# B&R Automation Studio project NAELD004C00R10L518F00 (part 27)

#### Act_Main.st
```iecst
(** 2019-07-03 **)
ACTION Act_Main:

	IF eStatOld <> eStat THEN
		fbDirCreate1(bEn := FALSE);
		fbDirCreate2(bEn := FALSE);
		fbFileRead1(bEn := FALSE);
		fbFileWrite1(bEn := FALSE);
		usiStep	:= 0;

		bFileNotFound			:= FALSE;
		bNewProduct				:= FALSE;
		bLastProductUnload		:= FALSE;
		bLastProductLeftInBffr	:= FALSE;

		sStatTxt	:= a_sStatText[eStat];

		eStatOld	:= eStat;

		eStatus		:= Busy;
	END_IF

	//Main
	CASE eStat OF

		BufferActIdle:
			eStatus	:= Idle;

		BufferActCreateDir:
			IF eStatus = Idle OR eStatus = Busy THEN

				eStatus	:= Busy;

				CASE usiStep OF
					0:
						fbDirCreate1(bEn := TRUE);
						IF fbDirCreate1.udiStatus = 0 THEN
							usiStep	:= 1;
						ELSIF fbDirCreate1.udiStatus < 65534 THEN
							eStatus		:= Error;

							IF fbDirCreate1.udiStatus = 1908 THEN
								udiStatus	:= 10000;	//Create User Directory Error
							ELSE
								udiStatus	:= fbDirCreate1.udiStatus;
							END_IF
						END_IF

					1:
						fbDirCreate2(bEn := TRUE);
						IF fbDirCreate2.udiStatus = 0 THEN
							eStatus	:= Done;
						ELSIF fbDirCreate2.udiStatus < 65534 THEN
							eStatus		:= Error;

							IF fbDirCreate2.udiStatus = 1908 THEN
								udiStatus	:= 10001;	//Create Retain Directory Error
							ELSE
								udiStatus	:= fbDirCreate2.udiStatus;
							END_IF
						END_IF

				END_CASE

			END_IF

		BufferActGetRetainBffr:
			IF eStatus = Idle OR eStatus = Busy THEN

				eStatus	:= Busy;

				fbFileRead1(bEn := TRUE);
				IF fbFileRead1.udiStatus = 0 THEN
					eStatus	:= Done;

					tyBffrParameter.diBffrTtlSlt	:= p_diBffrTtlSlt;
					tyBffrParameter.diSltCap		:= p_diSltCap;

					fBffrStat(ADR(p_tyBufferStat) , p_tyBuffer);
					fDispBffrDescending(ADR(p_tyDispBuffer) , tyBffrParameter , p_tyBuffer , p_dtCurrDT , DINT_TO_TIME(p_diCoolTm) , 0 , 1 , 2);

				ELSIF fbFileRead1.udiStatus < 65534 THEN
					eStatus	:= Error;

					IF fbFileRead1.udiStatus = 1900 THEN
						udiStatus	:= 10002;	//File Open Error While Reading Retain File
					ELSIF fbFileRead1.udiStatus = 1902 THEN
						udiStatus	:= 10003;	//File Read Error While Reading Retain File
					ELSIF fbFileRead1.udiStatus = 1904 THEN
						udiStatus	:= 10004;	//File Close Error While Reading Retain File
					ELSIF fbFileRead1.udiStatus = 1915 THEN
						eStatus			:= Done;
						bFileNotFound	:= TRUE;
					ELSE
						udiStatus	:= fbFileRead1.udiStatus;
					END_IF
				END_IF

			END_IF

		BufferActSetFull:
			IF eStatus = Idle OR eStatus = Busy THEN

				eStatus	:= Busy;

				CASE usiStep OF
					0:
						tyBffrParameter.bAscending		:= p_bAscending;
						tyBffrParameter.diBffrTtlSlt	:= p_diBffrTtlSlt;
						tyBffrParameter.diMaxSlt		:= p_diMaxSlt;
						tyBffrParameter.diMinSlt		:= p_diMinSlt;
						tyBffrParameter.diPitch			:= p_diPitch;
						tyBffrParameter.diSltCap		:= p_diSltCap;
						tyBffrParameter.a_bSkip			:= pa_bSkip;
						bFIFOOld						:= p_bFIFO;

						udiStatus	:= fBffrSetFull(ADR(p_tyBuffer) , tyBffrParameter , p_dtCurrDT , p_sBffrNm , p_sProdNm);

						IF udiStatus = 0 THEN
							usiStep	:= 1;

							fBffrStat(ADR(p_tyBufferStat) , p_tyBuffer);
							fDispBffrDescending(ADR(p_tyDispBuffer) , tyBffrParameter , p_tyBuffer , p_dtCurrDT , DINT_TO_TIME(p_diCoolTm) , 0 , 1 , 2);

						ELSE
							eStatus	:= Error;

						END_IF

					1:
						fbFileWrite1(bEn := TRUE);

						IF fbFileWrite1.udiStatus = 0 THEN
							eStatus	:= Done;
						ELSIF fbFileWrite1.udiStatus < 65534 THEN
							eStatus	:= Error;

							IF fbFileWrite1.udiStatus = 1900 THEN
								udiStatus	:= 10005;	//File Open Error While Setting Full Buffer
							ELSIF fbFileWrite1.udiStatus = 1901 THEN
								udiStatus	:= 10006;	//File Create Error While Setting Full Buffer
							ELSIF fbFileWrite1.udiStatus = 1903 THEN
								udiStatus	:= 10007;	//File Write Error While Setting Full Buffer
							ELSIF fbFileWrite1.udiStatus = 1904 THEN
								udiStatus	:= 10008;	//File Close Error While Setting Full Buffer
							ELSIF fbFileWrite1.udiStatus = 1914 THEN
								udiStatus	:= 10040;	//Directory Does Not Exist While Setting Full Buffer
							ELSE
								udiStatus	:= fbFileWrite1.udiStatus;
							END_IF
						END_IF

				END_CASE

			END_IF

		BufferActSetMty:
			IF eStatus = Idle OR eStatus = Busy THEN

				eStatus	:= Busy;

				CASE usiStep OF
					0:
						tyBffrParameter.bAscending		:= p_bAscending;
						tyBffrParameter.diBffrTtlSlt	:= p_diBffrTtlSlt;
						tyBffrParameter.diMaxSlt		:= p_diMaxSlt;
						tyBffrParameter.diMinSlt		:= p_diMinSlt;
						tyBffrParameter.diPitch			:= p_diPitch;
						tyBffrParameter.diSltCap		:= p_diSltCap;
						tyBffrParameter.a_bSkip			:= pa_bSkip;
						bFIFOOld						:= p_bFIFO;

						udiStatus	:= fBffrSetMty(ADR(p_tyBuffer) , tyBffrParameter , p_sBffrNm);

						IF udiStatus = 0 THEN
							usiStep	:= 1;

							fBffrStat(ADR(p_tyBufferStat) , p_tyBuffer);
							fDispBffrDescending(ADR(p_tyDispBuffer) , tyBffrParameter , p_tyBuffer , p_dtCurrDT , DINT_TO_TIME(p_diCoolTm) , 0 , 1 , 2);

						ELSE
							eStatus	:= Error;

						END_IF

					1:
						fbFileWrite1(bEn := TRUE);

						IF fbFileWrite1.udiStatus = 0 THEN
							eStatus	:= Done;
						ELSIF fbFileWrite1.udiStatus < 65534 THEN
							eStatus	:= Error;

							IF fbFileWrite1.udiStatus = 1900 THEN
								udiStatus	:= 10009;	//File Open Error While Setting Empty Buffer
							ELSIF fbFileWrite1.udiStatus = 1901 THEN
								udiStatus	:= 10010;	//File Create Error While Setting Empty Buffer
							ELSIF fbFileWrite1.udiStatus = 1903 THEN
								udiStatus	:= 10011;	//File Write Error While Setting Empty Buffer
							ELSIF fbFileWrite1.udiStatus = 1904 THEN
								udiStatus	:= 10012;	//File Close Error While Setting Empty Buffer
							ELSIF fbFileWrite1.udiStatus = 1914 THEN
								udiStatus	:= 10041;	//Directory Does Not Exist While Setting Empty Buffer
							ELSE
								udiStatus	:= fbFileWrite1.udiStatus;
							END_IF
						END_IF

				END_CASE

			END_IF

		BufferActLoad:
			IF eStatus = Idle OR eStatus = Busy THEN

				eStatus	:= Busy;

				CASE usiStep OF
					0:
						diCurrSlt	:= fLifterPosInUMToSltBtmMin(p_diLifterCurrPosInUM , p_diSltToSltInUM , p_diLifterBtmPosInUM);

						udiStatus	:= fBffrLoad(ADR(p_tyBuffer) , ADR(bNewProduct) , diCurrSlt , p_dtCurrDT , p_bGdBrdIn , p_sProdNm , p_sBarcode1 , p_sBarcode2);

						IF udiStatus = 0 THEN
							usiStep	:= 1;

							tyBffrParameter.diBffrTtlSlt	:= p_diBffrTtlSlt;
							tyBffrParameter.diSltCap		:= p_diSltCap;

							fBffrStat(ADR(p_tyBufferStat) , p_tyBuffer);
							fDispBffrDescending(ADR(p_tyDispBuffer) , tyBffrParameter , p_tyBuffer , p_dtCurrDT , DINT_TO_TIME(p_diCoolTm) , 0 , 1 , 2);

						ELSE
							eStatus	:= Error;

							IF udiStatus = 1010 THEN
								udiStatus	:= 10076;	//Loading Slot Is Not For Board
							ELSIF udiStatus = 1011 THEN
								udiStatus	:= 10077;	//Loading Slot Is Full Of Board
							ELSIF udiStatus = 1012 THEN
								udiStatus	:= 10078;	//Loading First Sub-Slot Is Not For Board
							ELSIF udiStatus	= 1013 THEN
								udiStatus	:= 10079;	//Loading Last Sub-Slot Have Board, Which Mean Slot Is Full Of Board
							ELSIF udiStatus = 1014 THEN
								udiStatus	:= 10080;	//Loading Last Sub-Slot Is Not For Board
							ELSIF udiStatus = 1015 THEN
								udiStatus	:= 10081;	//Loading Slot Is Full Of Board
							ELSIF udiStatus = 1001 THEN
								udiStatus	:= 10082;	//Loading Slot Is Skipped
							ELSIF udiStatus	= 1016 THEN
								udiStatus	:= 10083;	//Existing Board Status Is Different With Loading Board Status
							END_IF

						END_IF

					1:
						fbFileWrite1(bEn := TRUE);

						IF fbFileWrite1.udiStatus = 0 THEN
							eStatus	:= Done;
						ELSIF fbFileWrite1.udiStatus < 65534 THEN
							eStatus	:= Error;

							IF fbFileWrite1.udiStatus = 1900 THEN
								udiStatus	:= 10013;	//File Open Error While Loading Info To Buffer
							ELSIF fbFileWrite1.udiStatus = 1901 THEN
								udiStatus	:= 10014;	//File Create Error While Loading Info To Buffer
							ELSIF fbFileWrite1.udiStatus = 1903 THEN
								udiStatus	:= 10015;	//File Write Error While Loading Info To Buffer
							ELSIF fbFileWrite1.udiStatus = 1904 THEN
								udiStatus	:= 10016;	//File Close Error While Loading Info To Buffer
							ELSIF fbFileWrite1.udiStatus = 1914 THEN
								udiStatus	:= 10042;	//Directory Does Not Exist While Loading Info To Buffer
							ELSE
								udiStatus	:= fbFileWrite1.udiStatus;
							END_IF
						END_IF

				END_CASE

			END_IF

		BufferActLoadSltChk:
			IF eStatus = Idle OR eStatus = Busy THEN

				eStatus	:= Busy;

				CASE usiStep OF
					0:
						diCurrSlt	:= fLifterPosInUMToSltBtmMin(p_diLifterCurrPosInUM , p_diSltToSltInUM , p_diLifterBtmPosInUM);

						IF p_bNxtLoadSeq = TRUE AND p_bGdBrdIn = TRUE THEN
							diExpectedSlt	:= fBffrNxtLoadSeqGd(p_bAscending , p_tyBuffer);
						ELSIF p_bNxtLoadSeq = TRUE AND p_bGdBrdIn = FALSE THEN
							diExpectedSlt	:= fBffrNxtLoadSeqBad(p_bAscending , p_tyBuffer);
						ELSIF p_bNxtLoadSeq = FALSE AND p_bGdBrdIn = TRUE THEN
							diExpectedSlt	:= fBffrNxtLoadNearbyGd(diCurrSlt , p_tyBuffer);
						ELSE
							diExpectedSlt	:= fBffrNxtLoadNearbyBad(diCurrSlt , p_tyBuffer);
						END_IF

						IF diCurrSlt = diExpectedSlt THEN
							udiStatus	:= fBffrLoad(ADR(p_tyBuffer) , ADR(bNewProduct) , diCurrSlt , p_dtCurrDT , p_bGdBrdIn , p_sProdNm , p_sBarcode1 , p_sBarcode2);

							IF udiStatus = 0 THEN
								usiStep	:= 1;

								tyBffrParameter.diBffrTtlSlt	:= p_diBffrTtlSlt;
								tyBffrParameter.diSltCap		:= p_diSltCap;

								fBffrStat(ADR(p_tyBufferStat) , p_tyBuffer);
								fDispBffrDescending(ADR(p_tyDispBuffer) , tyBffrParameter , p_tyBuffer , p_dtCurrDT , DINT_TO_TIME(p_diCoolTm) , 0 , 1 , 2);

							ELSE
								eStatus	:= Error;

								IF udiStatus = 1010 THEN
									udiStatus	:= 10084;	//Loading Slot Is Not For Board
								ELSIF udiStatus = 1011 THEN
									udiStatus	:= 10085;	//Loading Slot Is Full Of Board
								ELSIF udiStatus = 1012 THEN
									udiStatus	:= 10086;	//Loading First Sub-Slot Is Not For Board
								ELSIF udiStatus	= 1013 THEN
									udiStatus	:= 10087;	//Loading Last Sub-Slot Have Board, Which Mean Slot Is Full Of Board
								ELSIF udiStatus = 1014 THEN
									udiStatus	:= 10088;	//Loading Last Sub-Slot Is Not For Board
								ELSIF udiStatus = 1015 THEN
									udiStatus	:= 10089;	//Loading Slot Is Full Of Board
								ELSIF udiStatus = 1001 THEN
									udiStatus	:= 10090;	//Loading Slot Is Skipped
								ELSIF udiStatus	= 1016 THEN
									udiStatus	:= 10091;	//Existing Board Status Is Different With Loading Board Status
								END_IF

							END_IF

						ELSE
							udiStatus	:= 10017;	//Wrong Slot Number To Load
							eStatus		:= Error;

						END_IF

					1:
						fbFileWrite1(bEn := TRUE);

						IF fbFileWrite1.udiStatus = 0 THEN
							eStatus	:= Done;
						ELSIF fbFileWrite1.udiStatus < 65534 THEN
							eStatus	:= Error;

							IF fbFileWrite1.udiStatus = 1900 THEN
								udiStatus	:= 10018;	//File Open Error While Loading Info To Buffer With Slot Check
							ELSIF fbFileWrite1.udiStatus = 1901 THEN
								udiStatus	:= 10019;	//File Create Error While Loading Info To Buffer With Slot Check
							ELSIF fbFileWrite1.udiStatus = 1903 THEN
								udiStatus	:= 10020;	//File Write Error While Loading Info To Buffer With Slot Check
							ELSIF fbFileWrite1.udiStatus = 1904 THEN
								udiStatus	:= 10021;	//File Close Error While Loading Info To Buffer With Slot Check
							ELSIF fbFileWrite1.udiStatus = 1914 THEN
								udiStatus	:= 10043;	//Directory Does Not Exist While Loading Info To Buffer With Slot Check
							ELSE
								udiStatus	:= fbFileWrite1.udiStatus;
							END_IF
						END_IF

				END_CASE

			END_IF

		BufferActUnload:
			IF eStatus = Idle OR eStatus = Busy THEN

				eStatus	:= Busy;

				CASE usiStep OF
					0:
						IF p_bLinkMcParamProdSelTopToBtm  AND p_bLinkProjLifterMagPlatform = FALSE THEN //TravLif with Top to Btm
							diCurrSlt	:= fLifterPosInUMToSltTopMin(p_diLifterCurrPosInUM , p_diSltToSltInUM , p_diLifterBtmPosInUM);
						ELSE
							diCurrSlt	:= fLifterPosInUMToSltBtmMin(p_diLifterCurrPosInUM , p_diSltToSltInUM , p_diLifterBtmPosInUM);
						END_IF

						udiStatus	:= fBffrUnload(ADR(tyBoardUnloadStat) , ADR(p_tyBuffer) , ADR(bLastProductUnload) , ADR(bLastProductLeftInBffr) , diCurrSlt);

						IF p_sCurrRcpNm = tyBoardUnloadStat.sProdNm THEN
							bLastProductUnload	:= FALSE;
						END_IF

						IF udiStatus = 0 THEN
							usiStep	:= 1;

							tyBffrParameter.diBffrTtlSlt	:= p_diBffrTtlSlt;
							tyBffrParameter.diSltCap		:= p_diSltCap;

							fBffrStat(ADR(p_tyBufferStat) , p_tyBuffer);
							fDispBffrDescending(ADR(p_tyDispBuffer) , tyBffrParameter , p_tyBuffer , p_dtCurrDT , DINT_TO_TIME(p_diCoolTm) , 0 , 1 , 2);

						ELSE
							eStatus	:= Error;

							IF udiStatus = 1000 THEN
								udiStatus	:= 10048;	//Unloading Slot Is Skipped While Unloading Buffer
							ELSIF udiStatus = 1003 THEN
								udiStatus	:= 10049;	//Unloading Slot Is Not For Board While Unloading Buffer
							ELSIF udiStatus = 1004 THEN
								udiStatus	:= 10050;	//Unloading Slot Board Is Not available While Unloading Buffer
							ELSIF udiStatus = 1005 THEN
								udiStatus	:= 10051;	//Unloading Last Sub Slot Is Not For Board While Unloading Buffer
							ELSIF udiStatus = 1006 THEN
								udiStatus	:= 10052;	//Unloading Last Sub Slot Has No Board While Unloading Buffer
							ELSIF udiStatus = 1007 THEN
								udiStatus	:= 10053;	//Board Quantity In Slot Is 0 While Unloading Buffer
							ELSIF udiStatus = 1008 THEN
								udiStatus	:= 10054;	//Board Capacity In Slot Is 0 While Unloading Buffer
							END_IF

						END_IF

					1:
						fbFileWrite1(bEn := TRUE);

						IF fbFileWrite1.udiStatus = 0 THEN
							eStatus	:= Done;
						ELSIF fbFileWrite1.udiStatus < 65534 THEN
							eStatus	:= Error;

							IF fbFileWrite1.udiStatus = 1900 THEN
								udiStatus	:= 10022;	//File Open Error While Unloading Info From Buffer
							ELSIF fbFileWrite1.udiStatus = 1901 THEN
								udiStatus	:= 10023;	//File Create Error While Unloading Info From Buffer
							ELSIF fbFileWrite1.udiStatus = 1903 THEN
								udiStatus	:= 10024;	//File Write Error While Unloading Info From Buffer
							ELSIF fbFileWrite1.udiStatus = 1904 THEN
								udiStatus	:= 10025;	//File Close Error While Unloading Info From Buffer
							ELSIF fbFileWrite1.udiStatus = 1914 THEN
								udiStatus	:= 10044;	//Directory Does Not Exist While Unloading Info From Buffer
							ELSE
								udiStatus	:= fbFileWrite1.udiStatus;
							END_IF
						END_IF

				END_CASE

			END_IF

		BufferActUnloadSltChk:
			IF eStatus = Idle OR eStatus = Busy THEN

				eStatus	:= Busy;

				CASE usiStep OF
					0:
						diCurrSlt	:= fLifterPosInUMToSltBtmMin(p_diLifterCurrPosInUM , p_diSltToSltInUM , p_diLifterBtmPosInUM);

						IF p_bFIFO = TRUE AND p_bGdBrdReq = TRUE THEN
							diExpectedSlt	:= fBffrNxtUnloadFIFOGd(p_tyBuffer , '');
						ELSIF p_bFIFO = TRUE AND p_bGdBrdReq = FALSE THEN
							diExpectedSlt	:= fBffrNxtUnloadFIFOBad(p_tyBuffer , '');
						ELSIF p_bFIFO = FALSE AND p_bGdBrdReq = TRUE THEN
							diExpectedSlt	:= fBffrNxtUnloadLIFOGd(p_tyBuffer , '');
						ELSE
							diExpectedSlt	:= fBffrNxtUnloadLIFOBad(p_tyBuffer , '');
						END_IF

						IF diCurrSlt = diExpectedSlt THEN
							udiStatus	:= fBffrUnload(ADR(tyBoardUnloadStat) , ADR(p_tyBuffer) , ADR(bLastProductUnload) , ADR(bLastProductLeftInBffr) , diCurrSlt);

							IF p_sCurrRcpNm = tyBoardUnloadStat.sProdNm THEN
								bLastProductUnload	:= FALSE;
							END_IF

							IF udiStatus = 0 THEN
								usiStep	:= 1;

								tyBffrParameter.diBffrTtlSlt	:= p_diBffrTtlSlt;
								tyBffrParameter.diSltCap		:= p_diSltCap;

								fBffrStat(ADR(p_tyBufferStat) , p_tyBuffer);
								fDispBffrDescending(ADR(p_tyDispBuffer) , tyBffrParameter , p_tyBuffer , p_dtCurrDT , DINT_TO_TIME(p_diCoolTm) , 0 , 1 , 2);

							ELSE
								eStatus	:= Error;

								IF udiStatus = 1000 THEN
									udiStatus	:= 10055;	//Unloading Slot Is Skipped While Unloading Buffer With Slot Check
								ELSIF udiStatus = 1003 THEN
									udiStatus	:= 10056;	//Unloading Slot Is Not For Board While Unloading Buffer With Slot Check
								ELSIF udiStatus = 1004 THEN
									udiStatus	:= 10057;	//Unloading Slot Board Is Not available While Unloading Buffer With Slot Check
								ELSIF udiStatus = 1005 THEN
									udiStatus	:= 10058;	//Unloading Last Sub Slot Is Not For Board While Unloading Buffer With Slot Check
								ELSIF udiStatus = 1006 THEN
									udiStatus	:= 10059;	//Unloading Last Sub Slot Has No Board While Unloading Buffer With Slot Check
								ELSIF udiStatus = 1007 THEN
									udiStatus	:= 10060;	//Board Quantity In Slot Is 0 While Unloading Buffer With Slot Check
								ELSIF udiStatus = 1008 THEN
									udiStatus	:= 10061;	//Board Capacity In Slot Is 0 While Unloading Buffer With Slot Check
								END_IF

							END_IF

						ELSE
							udiStatus	:= 10026;	//Wrong Slot Number To Unload
							eStatus		:= Error;

						END_IF

					1:
						fbFileWrite1(bEn := TRUE);

						IF fbFileWrite1.udiStatus = 0 THEN
							eStatus	:= Done;
						ELSIF fbFileWrite1.udiStatus < 65534 THEN
							eStatus	:= Error;

							IF fbFileWrite1.udiStatus = 1900 THEN
								udiStatus	:= 10027;	//File Open Error While Unloading Info From Buffer With Slot Check
							ELSIF fbFileWrite1.udiStatus = 1901 THEN
								udiStatus	:= 10028;	//File Create Error While Unloading Info From Buffer With Slot Check
							ELSIF fbFileWrite1.udiStatus = 1903 THEN
								udiStatus	:= 10029;	//File Write Error While Unloading Info From Buffer With Slot Check
							ELSIF fbFileWrite1.udiStatus = 1904 THEN
								udiStatus	:= 10030;	//File Close Error While Unloading Info From Buffer With Slot Check
							ELSIF fbFileWrite1.udiStatus = 1914 THEN
								udiStatus	:= 10045;	//Directory Does Not Exist While Unloading Info From Buffer With Slot Check
							ELSE
								udiStatus	:= fbFileWrite1.udiStatus;
							END_IF
						END_IF

				END_CASE

			END_IF

		BufferActUnloadCoolChk:
			IF eStatus = Idle OR eStatus = Busy THEN

				eStatus	:= Busy;

				CASE usiStep OF
					0:
						diCurrSlt	:= fLifterPosInUMToSltBtmMin(p_diLifterCurrPosInUM , p_diSltToSltInUM , p_diLifterBtmPosInUM);

						bCoolNotRdy	:= NOT fBffrChkCoolTmRdy(diCurrSlt, p_dtCurrDT, DINT_TO_TIME(p_diCoolTm), p_tyBuffer);

						IF bCoolNotRdy = FALSE THEN
							udiStatus	:= fBffrUnload(ADR(tyBoardUnloadStat) , ADR(p_tyBuffer) , ADR(bLastProductUnload) , ADR(bLastProductLeftInBffr) , diCurrSlt);

							IF p_sCurrRcpNm = tyBoardUnloadStat.sProdNm THEN
								bLastProductUnload	:= FALSE;
							END_IF

							IF udiStatus = 0 THEN
								usiStep	:= 1;

								tyBffrParameter.diBffrTtlSlt	:= p_diBffrTtlSlt;
								tyBffrParameter.diSltCap		:= p_diSltCap;

								fBffrStat(ADR(p_tyBufferStat) , p_tyBuffer);
								fDispBffrDescending(ADR(p_tyDispBuffer) , tyBffrParameter , p_tyBuffer , p_dtCurrDT , DINT_TO_TIME(p_diCoolTm) , 0 , 1 , 2);

							ELSE
								eStatus	:= Error;

								IF udiStatus = 1000 THEN
									udiStatus	:= 10062;	//Unloading Slot Is Skipped While Unloading Buffer With Cool Check
								ELSIF udiStatus = 1003 THEN
									udiStatus	:= 10063;	//Unloading Slot Is Not For Board While Unloading Buffer With Cool Check
								ELSIF udiStatus = 1004 THEN
									udiStatus	:= 10064;	//Unloading Slot Board Is Not available While Unloading Buffer With Cool Check
								ELSIF udiStatus = 1005 THEN
									udiStatus	:= 10065;	//Unloading Last Sub Slot Is Not For Board While Unloading Buffer With Cool Check
								ELSIF udiStatus = 1006 THEN
									udiStatus	:= 10066;	//Unloading Last Sub Slot Has No Board While Unloading Buffer With Cool Check
								ELSIF udiStatus = 1007 THEN
									udiStatus	:= 10067;	//Board Quantity In Slot Is 0 While Unloading Buffer With Cool Check
								ELSIF udiStatus = 1008 THEN
									udiStatus	:= 10068;	//Board Capacity In Slot Is 0 While Unloading Buffer With Cool Check
								END_IF

							END_IF

						ELSE
							eStatus	:= Done;

						END_IF

					1:
						fbFileWrite1(bEn := TRUE);

						IF fbFileWrite1.udiStatus = 0 THEN
							eStatus	:= Done;
						ELSIF fbFileWrite1.udiStatus < 65534 THEN
							eStatus	:= Error;

							IF fbFileWrite1.udiStatus = 1900 THEN
								udiStatus	:= 10031;	//File Open Error While Unloading Info From Buffer With Cooling Time Check
							ELSIF fbFileWrite1.udiStatus = 1901 THEN
								udiStatus	:= 10032;	//File Create Error While Unloading Info From Buffer With Cooling Time Check
							ELSIF fbFileWrite1.udiStatus = 1903 THEN
								udiStatus	:= 10033;	//File Write Error While Unloading Info From Buffer With Cooling Time Check
							ELSIF fbFileWrite1.udiStatus = 1904 THEN
								udiStatus	:= 10034;	//File Close Error While Unloading Info From Buffer With Cooling Time Check
							ELSIF fbFileWrite1.udiStatus = 1914 THEN
								udiStatus	:= 10046;	//Directory Does Not Exist While Unloading Info From Buffer With Cooling Time Check
							ELSE
								udiStatus	:= fbFileWrite1.udiStatus;
							END_IF
						END_IF

				END_CASE

			END_IF

		BufferActUnloadSltChkCoolChk:
			IF eStatus = Idle OR eStatus = Busy THEN

				eStatus	:= Busy;

				CASE usiStep OF
					0:
						diCurrSlt	:= fLifterPosInUMToSltBtmMin(p_diLifterCurrPosInUM , p_diSltToSltInUM , p_diLifterBtmPosInUM);

						IF p_bFIFO = TRUE AND p_bGdBrdReq = TRUE THEN
							diExpectedSlt	:= fBffrNxtUnloadFIFOGd(p_tyBuffer , '');
						ELSIF p_bFIFO = TRUE AND p_bGdBrdReq = FALSE THEN
							diExpectedSlt	:= fBffrNxtUnloadFIFOBad(p_tyBuffer , '');
						ELSIF p_bFIFO = FALSE AND p_bGdBrdReq = TRUE THEN
							diExpectedSlt	:= fBffrNxtUnloadLIFOGd(p_tyBuffer , '');
						ELSE
							diExpectedSlt	:= fBffrNxtUnloadLIFOBad(p_tyBuffer , '');
						END_IF

						IF diCurrSlt = diExpectedSlt THEN
							bCoolNotRdy	:= NOT fBffrChkCoolTmRdy(diCurrSlt, p_dtCurrDT, DINT_TO_TIME(p_diCoolTm), p_tyBuffer);

							IF bCoolNotRdy = FALSE THEN
								udiStatus	:= fBffrUnload(ADR(tyBoardUnloadStat) , ADR(p_tyBuffer) , ADR(bLastProductUnload) , ADR(bLastProductLeftInBffr) , diCurrSlt);

								IF p_sCurrRcpNm = tyBoardUnloadStat.sProdNm THEN
									bLastProductUnload	:= FALSE;
								END_IF

								IF udiStatus = 0 THEN
									usiStep	:= 1;

									tyBffrParameter.diBffrTtlSlt	:= p_diBffrTtlSlt;
									tyBffrParameter.diSltCap		:= p_diSltCap;

									fBffrStat(ADR(p_tyBufferStat) , p_tyBuffer);
									fDispBffrDescending(ADR(p_tyDispBuffer) , tyBffrParameter , p_tyBuffer , p_dtCurrDT , DINT_TO_TIME(p_diCoolTm) , 0 , 1 , 2);

								ELSE
									eStatus	:= Error;

									IF udiStatus = 1000 THEN
										udiStatus	:= 10069;	//Unloading Slot Is Skipped While Unloading Buffer With Cool & Slot Check
									ELSIF udiStatus = 1003 THEN
										udiStatus	:= 10070;	//Unloading Slot Is Not For Board While Unloading Buffer With Cool & Slot Check
									ELSIF udiStatus = 1004 THEN
										udiStatus	:= 10071;	//Unloading Slot Board Is Not available While Unloading Buffer With Cool & Slot Check
									ELSIF udiStatus = 1005 THEN
										udiStatus	:= 10072;	//Unloading Last Sub Slot Is Not For Board While Unloading Buffer With Cool & Slot Check
									ELSIF udiStatus = 1006 THEN
										udiStatus	:= 10073;	//Unloading Last Sub Slot Has No Board While Unloading Buffer With Cool & Slot Check
									ELSIF udiStatus = 1007 THEN
										udiStatus	:= 10074;	//Board Quantity In Slot Is 0 While Unloading Buffer With Cool & Slot Check
									ELSIF udiStatus = 1008 THEN
										udiStatus	:= 10075;	//Board Capacity In Slot Is 0 While Unloading Buffer With Cool & Slot Check
									END_IF

								END_IF

							ELSE
								eStatus	:= Done;

							END_IF

						ELSE
							udiStatus	:= 10035;	//Wrong Slot Number To Unload With Cooling Time Check
							eStatus		:= Error;

						END_IF

					1:
						fbFileWrite1(bEn := TRUE);

						IF fbFileWrite1.udiStatus = 0 THEN
							eStatus	:= Done;
						ELSIF fbFileWrite1.udiStatus < 65534 THEN
							eStatus	:= Error;

							IF fbFileWrite1.udiStatus = 1900 THEN
								udiStatus	:= 10036;	//File Open Error While Unloading Info From Buffer With Slot Check And Cooling Time Check
							ELSIF fbFileWrite1.udiStatus = 1901 THEN
								udiStatus	:= 10037;	//File Create Error While Unloading Info From Buffer With Slot Check And Cooling Time Check
							ELSIF fbFileWrite1.udiStatus = 1903 THEN
								udiStatus	:= 10038;	//File Write Error While Unloading Info From Buffer With Slot Check And Cooling Time Check
							ELSIF fbFileWrite1.udiStatus = 1904 THEN
								udiStatus	:= 10039;	//File Close Error While Unloading Info From Buffer With Slot Check And Cooling Time Check
							ELSIF fbFileWrite1.udiStatus = 1914 THEN
								udiStatus	:= 10047;	//Directory Does Not Exist While Unloading Info From Buffer With Slot Check And Cooling Time Check
							ELSE
								udiStatus	:= fbFileWrite1.udiStatus;
							END_IF
						END_IF

				END_CASE

			END_IF

		BufferActNxtLoad:
			IF eStatus = Idle OR eStatus = Busy THEN

				diCurrSlt	:= fLifterPosInUMToSltBtmMin(p_diLifterCurrPosInUM , p_diSltToSltInUM , p_diLifterBtmPosInUM);

				IF p_bNxtLoadSeq = TRUE THEN
					diNxtLoadSlt	:= fBffrNxtLoadSeqAny(p_bAscending , p_tyBuffer);
				ELSE
					diNxtLoadSlt	:= fBffrNxtLoadNearbyAny(diCurrSlt , p_tyBuffer);
				END_IF

				eStatus	:= Done;

			END_IF

		BufferActNxtLoadGd:
			IF eStatus = Idle OR eStatus = Busy THEN

				diCurrSlt	:= fLifterPosInUMToSltBtmMin(p_diLifterCurrPosInUM , p_diSltToSltInUM , p_diLifterBtmPosInUM);

				IF p_bNxtLoadSeq = TRUE THEN
					diNxtLoadSlt	:= fBffrNxtLoadSeqGd(p_bAscending , p_tyBuffer);
				ELSE
					diNxtLoadSlt	:= fBffrNxtLoadNearbyGd(diCurrSlt , p_tyBuffer);
				END_IF

				eStatus	:= Done;

			END_IF

		BufferActNxtLoadBad:
			IF eStatus = Idle OR eStatus = Busy THEN

				diCurrSlt	:= fLifterPosInUMToSltBtmMin(p_diLifterCurrPosInUM , p_diSltToSltInUM , p_diLifterBtmPosInUM);

				IF p_bNxtLoadSeq = TRUE THEN
					diNxtLoadSlt	:= fBffrNxtLoadSeqBad(p_bAscending , p_tyBuffer);
				ELSE
					diNxtLoadSlt	:= fBffrNxtLoadNearbyBad(diCurrSlt , p_tyBuffer);
				END_IF

				eStatus	:= Done;

			END_IF

		BufferActNxtUnload:
			IF eStatus = Idle OR eStatus = Busy THEN

				IF p_bFIFO = TRUE THEN
					diNxtUnloadSlt	:= fBffrNxtUnloadFIFOAny(p_tyBuffer , '');
				ELSE
					diNxtUnloadSlt	:= fBffrNxtUnloadLIFOAny(p_tyBuffer , '');
				END_IF

				eStatus	:= Done;

			END_IF

		BufferActNxtUnloadGd:
			IF eStatus = Idle OR eStatus = Busy THEN

				IF p_bFIFO = TRUE THEN
					diNxtUnloadSlt	:= fBffrNxtUnloadFIFOGd(p_tyBuffer , '');
				ELSE
					diNxtUnloadSlt	:= fBffrNxtUnloadLIFOGd(p_tyBuffer , '');
				END_IF

				eStatus	:= Done;

			END_IF

		BufferActNxtUnloadBad:
			IF eStatus = Idle OR eStatus = Busy THEN

				IF p_bFIFO = TRUE THEN
					diNxtUnloadSlt	:= fBffrNxtUnloadFIFOBad(p_tyBuffer , '');
				ELSE
					diNxtUnloadSlt	:= fBffrNxtUnloadLIFOBad(p_tyBuffer , '');
				END_IF

				eStatus	:= Done;

			END_IF

		BufferActChkCoolTm:
			diCurrSlt	:= fLifterPosInUMToSltBtmMin(p_diLifterCurrPosInUM , p_diSltToSltInUM , p_diLifterBtmPosInUM);

			bCoolNotRdy	:= NOT fBffrChkCoolTmRdy(diCurrSlt, p_dtCurrDT, DINT_TO_TIME(p_diCoolTm), p_tyBuffer);

			eStatus	:= Done;

		BufferActChkCoolBrdAny:
			diCoolBrdAny	:= fBffrChkCoolBrdAny(p_dtCurrDT, DINT_TO_TIME(p_diCoolTm), p_tyBuffer);

			eStatus	:= Done;

		BufferActChkCoolBrdGd:
			diCoolBrdGd		:= fBffrChkCoolBrdGd(p_dtCurrDT, DINT_TO_TIME(p_diCoolTm), p_tyBuffer);

			eStatus	:= Done;

		BufferActChkCoolBrdBad:
			diCoolBrdBad	:= fBffrChkCoolBrdBad(p_dtCurrDT, DINT_TO_TIME(p_diCoolTm), p_tyBuffer);

			eStatus	:= Done;

		BufferActRstBffr:
			IF eStatus = Idle OR eStatus = Busy THEN

				tyBffrParameter.diBffrTtlSlt	:= p_diBffrTtlSlt;
				tyBffrParameter.diSltCap		:= p_diSltCap;

				memset(ADR(p_tyBuffer) , 0 , SIZEOF(p_tyBuffer));
				fBffrStat(ADR(p_tyBufferStat) , p_tyBuffer);
				fDispBffrDescending(ADR(p_tyDispBuffer) , tyBffrParameter , p_tyBuffer , p_dtCurrDT , DINT_TO_TIME(p_diCoolTm) , 0 , 1 , 2);

				eStatus	:= Done;

			END_IF

		BufferActSetCoolFan:
			IF eStatus = Idle OR eStatus = Busy THEN

				bCoolFanCtrl	:= TRUE;
				eStatus			:= Done;

			END_IF

		BufferActRstCoolFan:
			IF eStatus = Idle OR eStatus = Busy THEN

				bCoolFanCtrl	:= FALSE;
				eStatus			:= Done;

			END_IF

		BufferActBGStartBffrSetFull:
			IF eStatus = Idle OR eStatus = Busy THEN

				bBffrSetFull	:= TRUE;
				bBffrSetMty		:= FALSE;
				eStatus			:= Done;

			END_IF

		BufferActBGStartBffrSetMty:
			IF eStatus = Idle OR eStatus = Busy THEN

				bBffrSetFull	:= FALSE;
				bBffrSetMty		:= TRUE;
				eStatus			:= Done;

			END_IF

		BufferActBGStopBffrSet:
			IF eStatus = Idle OR eStatus = Busy THEN

				bBffrSetFull	:= FALSE;
				bBffrSetMty		:= FALSE;
				eStatus			:= Done;

			END_IF

		BufferActBGStartUpdtSen:
			IF eStatus = Idle OR eStatus = Busy THEN

				bUpdateSensor	:= TRUE;
				eStatus			:= Done;

			END_IF

		BufferActBGStopUpdtSen:
			IF eStatus = Idle OR eStatus = Busy THEN

				bUpdateSensor	:= FALSE;
				eStatus			:= Done;

			END_IF

		BufferActBGStartUpdtDisplay:
			IF eStatus = Idle OR eStatus = Busy THEN

				bUpdtDisplay	:= TRUE;
				eStatus			:= Done;

			END_IF

		BufferActBGStopUpdtDisplay:
			IF eStatus = Idle OR eStatus = Busy THEN

				bUpdtDisplay	:= FALSE;
				eStatus			:= Done;

			END_IF

		BufferActBGStartCoolFan:
			IF eStatus = Idle OR eStatus = Busy THEN

				bCoolFanRun	:= TRUE;
				eStatus		:= Done;

			END_IF

		BufferActBGStopCoolFan:
			IF eStatus = Idle OR eStatus = Busy THEN

				bCoolFanRun	:= FALSE;
				eStatus		:= Done;

			END_IF

	END_CASE

END_ACTION
```

#### Init.st
```iecst
(** 2019-06-07 **)
PROGRAM _INIT

	(* Always Change If Project Change *)

	//Pass Address To Global Address For External Use
	//Action, State & Status
	p_Buffer2Stat		:= ADR(eStat);
	p_Buffer2Status		:= ADR(eStatus);
	p_Buffer2StatTxt	:= ADR(sStatTxt);

	//Alarm
	p_Buffer2AlmData	:= ADR(tyAlmData);

	//Output
	p_Buffer2NxtLoadSlt				:= ADR(diNxtLoadSlt);
	p_Buffer2NxtUnloadSlt			:= ADR(diNxtUnloadSlt);
	p_Buffer2CoolBrdAny				:= ADR(diCoolBrdAny);
	p_Buffer2CoolBrdGd				:= ADR(diCoolBrdGd);
	p_Buffer2CoolBrdBad				:= ADR(diCoolBrdBad);
	p_Buffer2CoolNotRdy				:= ADR(bCoolNotRdy);
	p_Buffer2Bffr					:= ADR(tyBuffer);
	p_Buffer2DispBffr				:= ADR(tyDispBuffer);
	p_Buffer2BffrStat				:= ADR(tyBufferStat);
	p_Buffer2BrdUnloadStat			:= ADR(tyBoardUnloadStat);
	p_Buffer2FileNotFound			:= ADR(bFileNotFound);
	p_Buffer2CoolFanCtrl			:= ADR(bCoolFanCtrl);
	p_Buffer2MagPresent				:= ADR(bMagPresent);
	p_Buffer2MagPresentTm			:= ADR(dtMagPresentTm);
	p_Buffer2NewProduct				:= ADR(bNewProduct);
	p_Buffer2LastProductUnload		:= ADR(bLastProductUnload);
	p_Buffer2LastProductLeftInBffr	:= ADR(bLastProductLeftInBffr);
	p_Buffer2ParamDiff				:= ADR(bParamDiff);
	p_Buffer2MagRemoved				:= ADR(bMagRemoved);
	p_Buffer2FIFOOld				:= ADR(bFIFOOld);

	//Svy Hermes
	p_Buffer2SlotNo					:= ADR(diCurrSltHermes);

	(* Always Change If Project Change *)

END_PROGRAM
```

### Program Logical/Buffer/Buffer3 (IEC) - 1.00.0 - NtBuffer v5.00.0 , NtFileIO v5.00.0

#### Local.var
```iecst
(*2019-06-07*)
(**)
(*Local Action, State & Status*)
VAR
	eAct : eBufferAction := BufferActIdle;
	eStat : eBufferAction := BufferActIdle;
	eStatus : eFBStatus := Idle;
	udiStatus : UDINT := 0;
	sStatTxt : STRING[200] := '';
	a_sStatText : ARRAY[0..50] OF STRING[200] := ['Idling','Creating Directory','Getting Retained Buffer Data','Setting Buffer Full','Setting Buffer Empty','Loading Board','Loading Board With Slot Check','Unloading Board','Unloading Board With Slot Check','Unloading Board With Cooling Time Check','Unloading Board With Slot Check And Cooling Time Check','Getting Next Load Board Slot Number','Getting Next Load Good Board Slot Number','Getting Next Load Bad Board Slot Number','Getting Next Unload Board Slot Number','Getting Next Unload Good Board Slot Number','Getting Next Unload Bad Board Slot Number','Checking Cooling Time','Checking Cooling Board','Checking Cooling Good Board','Checking Cooling Bad Board','Resetting Buffer','Turning On Cooling Fan','Turning Off Cooling Fan','Background Starting Buffer Set Full','Background Starting Buffer Set Empty','Background Stopping Buffer Set','Background Starting Update Sensor','Background Stopping Update Sensor','Background Starting Update Display','Background Stopping Update Display','Background Starting Cooling Fan','Background Stopping Cooling Fan',18('')];
END_VAR
(**)
(*Local Alarm*)
VAR
	tyAlmData : tyAlmDat;
	a_tyAlmText : ARRAY[10000..10099] OF tyAlmTxt := [(sAlmText:='Create User Directory Error',sRcyText:='An Error Occurred While Attempting To Create User Directory. Please Contact Nutek For A Possible Solution'),(sAlmText:='Create Retain Directory Error',sRcyText:='An Error Occurred While Attempting To Create Retain Directory. Please Contact Nutek For A Possible Solution'),(sAlmText:='File Open Error While Reading Retain File',sRcyText:='An Error Was Encountered While Trying To Open File. Please Contact Nutek For A Possible Solution.'),(sAlmText:='File Read Error While Reading Retain File',sRcyText:='An Error Was Encountered While Trying To Read File. Please Contact Nutek For A Possible Solution.'),(sAlmText:='File Close Error While Reading Retain File',sRcyText:='An Error Was Encountered While Trying To Close File. Please Contact Nutek For A Possible Solution.'),(sAlmText:='File Open Error While Setting Full Buffer',sRcyText:='An Error Was Encountered While Trying To Open File. Please Contact Nutek For A Possible Solution.'),(sAlmText:='File Create Error While Setting Full Buffer',sRcyText:='An Error Was Encountered While Trying To Create File. Please Contact Nutek For A Possible Solution.'),(sAlmText:='File Write Error While Setting Full Buffer',sRcyText:='An Error Was Encountered While Trying To Write File. Please Contact Nutek For A Possible Solution.'),(sAlmText:='File Close Error While Setting Full Buffer',sRcyText:='An Error Was Encountered While Trying To Close File. Please Contact Nutek For A Possible Solution.'),(sAlmText:='File Open Error While Setting Empty Buffer',sRcyText:='An Error Was Encountered While Trying To Open File. Please Contact Nutek For A Possible Solution.'),(sAlmText:='File Create Error While Setting Empty Buffer',sRcyText:='An Error Was Encountered While Trying To Create File. Please Contact Nutek For A Possible Solution.'),(sAlmText:='File Write Error While Setting Empty Buffer',sRcyText:='An Error Was Encountered While Trying To Write File. Please Contact Nutek For A Possible Solution.'),(sAlmText:='File Close Error While Setting Empty Buffer',sRcyText:='An Error Was Encountered While Trying To Close File. Please Contact Nutek For A Possible Solution.'),(sAlmText:='File Open Error While Loading Info To Buffer',sRcyText:='An Error Was Encountered While Trying To Open File. Please Contact Nutek For A Possible Solution.'),(sAlmText:='File Create Error While Loading Info To Buffer',sRcyText:='An Error Was Encountered While Trying To Create File. Please Contact Nutek For A Possible Solution.'),(sAlmText:='File Write Error While Loading Info To Buffer',sRcyText:='An Error Was Encountered While Trying To Write File. Please Contact Nutek For A Possible Solution.'),(sAlmText:='File Close Error While Loading Info To Buffer',sRcyText:='An Error Was Encountered While Trying To Close File. Please Contact Nutek For A Possible Solution.'),(sAlmText:='Wrong Slot Number To Load',sRcyText:='Invalid Slot to Load The Board.'),(sAlmText:='File Open Error While Loading Info To Buffer With Slot Check',sRcyText:='An Error Was Encountered While Trying To Open File. Please Contact Nutek For A Possible Solution.'),(sAlmText:='File Create Error While Loading Info To Buffer With Slot Check',sRcyText:='An Error Was Encountered While Trying To Create File. Please Contact Nutek For A Possible Solution.'),(sAlmText:='File Write Error While Loading Info To Buffer With Slot Check',sRcyText:='An Error Was Encountered While Trying To Write File. Please Contact Nutek For A Possible Solution.'),(sAlmText:='File Close Error While Loading Info To Buffer With Slot Check',sRcyText:='An Error Was Encountered While Trying To Close File. Please Contact Nutek For A Possible Solution.'),(sAlmText:='File Open Error While Unloading Info From Buffer',sRcyText:='An Error Was Encountered While Trying To Open File. Please Contact Nutek For A Possible Solution.'),(sAlmText:='File Create Error While Unloading Info From Buffer',sRcyText:='An Error Was Encountered While Trying To Create File. Please Contact Nutek For A Possible Solution.'),(sAlmText:='File Write Error While Unloading Info From Buffer',sRcyText:='An Error Was Encountered While Trying To Write File. Please Contact Nutek For A Possible Solution.'),(sAlmText:='File Close Error While Unloading Info From Buffer',sRcyText:='An Error Was Encountered While Trying To Close File. Please Contact Nutek For A Possible Solution.'),(sAlmText:='Wrong Slot Number To Unload',sRcyText:='Invalid Slot to Unload The Board.'),(sAlmText:='File Open Error While Unloading Info From Buffer With Slot Check',sRcyText:='An Error Was Encountered While Trying To Open File. Please Contact Nutek For A Possible Solution.'),(sAlmText:='File Create Error While Unloading Info From Buffer With Slot Check',sRcyText:='An Error Was Encountered While Trying To Create File. Please Contact Nutek For A Possible Solution.'),(sAlmText:='File Write Error While Unloading Info From Buffer With Slot Check',sRcyText:='An Error Was Encountered While Trying To Write File. Please Contact Nutek For A Possible Solution.'),(sAlmText:='File Close Error While Unloading Info From Buffer With Slot Check',sRcyText:='An Error Was Encountered While Trying To Close File. Please Contact Nutek For A Possible Solution.'),(sAlmText:='File Open Error While Unloading Info From Buffer With Cooling Time Check',sRcyText:='An Error Was Encountered While Trying To Open File. Please Contact Nutek For A Possible Solution.'),(sAlmText:='File Create Error While Unloading Info From Buffer With Cooling Time Check',sRcyText:='An Error Was Encountered While Trying To Create File. Please Contact Nutek For A Possible Solution.'),(sAlmText:='File Write Error While Unloading Info From Buffer With Cooling Time Check',sRcyText:='An Error Was Encountered While Trying To Write File. Please Contact Nutek For A Possible Solution.'),(sAlmText:='File Close Error While Unloading Info From Buffer With Cooling Time Check',sRcyText:='An Error Was Encountered While Trying To Close File. Please Contact Nutek For A Possible Solution.'),(sAlmText:='Wrong Slot Number To Unload With Cooling Time Check',sRcyText:='Invalid Slot to Unload The Board with Cooling Time Check.'),(sAlmText:='File Open Error While Unloading Info From Buffer With Slot Check And Cooling Time Check',sRcyText:='An Error Was Encountered While Trying To Open File. Please Contact Nutek For A Possible Solution.'),(sAlmText:='File Create Error While Unloading Info From Buffer With Slot Check And Cooling Time Check',sRcyText:='An Error Was Encountered While Trying To Create File. Please Contact Nutek For A Possible Solution.'),(sAlmText:='File Write Error While Unloading Info From Buffer With Slot Check And Cooling Time Check',sRcyText:='An Error Was Encountered While Trying To Write File. Please Contact Nutek For A Possible Solution.'),(sAlmText:='File Close Error While Unloading Info From Buffer With Slot Check And Cooling Time Check',sRcyText:='An Error Was Encountered While Trying To Close File. Please Contact Nutek For A Possible Solution.'),(sAlmText:='Directory Does Not Exist While Setting Full Buffer',sRcyText:='The Directory Does Not Exist. Please Contact Nutek For A Possible Solution.'),(sAlmText:='Directory Does Not Exist While Setting Empty Buffer',sRcyText:='The Directory Does Not Exist. Please Contact Nutek For A Possible Solution.'),(sAlmText:='Directory Does Not Exist While Loading Info To Buffer',sRcyText:='The Directory Does Not Exist. Please Contact Nutek For A Possible Solution.'),(sAlmText:='Directory Does Not Exist While Loading Info To Buffer With Slot Check',sRcyText:='The Directory Does Not Exist. Please Contact Nutek For A Possible Solution.'),(sAlmText:='Directory Does Not Exist While Unloading Info From Buffer',sRcyText:='The Directory Does Not Exist. Please Contact Nutek For A Possible Solution.'),(sAlmText:='Directory Does Not Exist While Unloading Info From Buffer With Slot Check',sRcyText:='The Directory Does Not Exist. Please Contact Nutek For A Possible Solution.'),(sAlmText:='Directory Does Not Exist While Unloading Info From Buffer With Cooling Time Check',sRcyText:='The Directory Does Not Exist. Please Contact Nutek For A Possible Solution.'),(sAlmText:='Directory Does Not Exist While Unloading Info From Buffer With Slot Check And Cooling Time Check',sRcyText:='The Directory Does Not Exist. Please Contact Nutek For A Possible Solution.'),(sAlmText:='Unloading Slot Is Skipped While Unloading Buffer',sRcyText:='Unload From Wrong Slot (Skip Slot).'),(sAlmText:='Unloading Slot Is Not For Board While Unloading Buffer',sRcyText:='Unload From Wrong Slot (Not For Board).'),(sAlmText:='Unloading Slot Board Is Not Available While Unloading Buffer',sRcyText:='Unload From Wrong Slot (Board Is Not Available).'),(sAlmText:='Unloading Last Sub Slot Is Not For Board While Unloading Buffer',sRcyText:='Unload From Wrong Slot (Last Sub Slot Is Not For Board).'),(sAlmText:='Unloading Last Sub Slot Has No Board While Unloading Buffer',sRcyText:='Unload From Wrong Slot (Last Sub Slot Has No Board).'),(sAlmText:='Board Quantity In Slot Is 0 While Unloading Buffer',sRcyText:='Unload From Wrong Slot (Board Quantity In Slot = 0).'),(sAlmText:='Board Capacity In Slot Is 0 While Unloading Buffer',sRcyText:='Unload From Wrong Slot (Board Capacity In Slot = 0).'),(sAlmText:='Unloading Slot Is Skipped While Unloading Buffer With Slot Check',sRcyText:='Unload From Wrong Slot (Skip Slot).'),(sAlmText:='Unloading Slot Is Not For Board While Unloading Buffer With Slot Check',sRcyText:='Unload From Wrong Slot (Not For Board).'),(sAlmText:='Unloading Slot Board Is Not available While Unloading Buffer With Slot Check',sRcyText:='Unload From Wrong Slot (Board Is Not Available).'),(sAlmText:='Unloading Last Sub Slot Is Not For Board While Unloading Buffer With Slot Check',sRcyText:='Unload From Wrong Slot (Last Sub Slot Is Not For Board).'),(sAlmText:='Unloading Last Sub Slot Has No Board While Unloading Buffer With Slot Check',sRcyText:='Unload From Wrong Slot (Last Sub Slot Has No Board).'),(sAlmText:='Board Quantity In Slot Is 0 While Unloading Buffer With Slot Check',sRcyText:='Unload From Wrong Slot (Board Quantity In Slot = 0).'),(sAlmText:='Board Capacity In Slot Is 0 While Unloading Buffer With Slot Check',sRcyText:='Unload From Wrong Slot (Board Capacity In Slot = 0).'),(sAlmText:='Unloading Slot Is Skipped While Unloading Buffer With Cool Check',sRcyText:='Unload From Wrong Slot (Skip Slot).'),(sAlmText:='Unloading Slot Is Not For Board While Unloading Buffer With Cool Check',sRcyText:='Unload From Wrong Slot (Not For Board).'),(sAlmText:='Unloading Slot Board Is Not available While Unloading Buffer With Cool Check',sRcyText:='Unload From Wrong Slot (Board Is Not Available).'),(sAlmText:='Unloading Last Sub Slot Is Not For Board While Unloading Buffer With Cool Check',sRcyText:='Unload From Wrong Slot (Last Sub Slot Is Not For Board).'),(sAlmText:='Unloading Last Sub Slot Has No Board While Unloading Buffer With Cool Check',sRcyText:='Unload From Wrong Slot (Last Sub Slot Has No Board).'),(sAlmText:='Board Quantity In Slot Is 0 While Unloading Buffer With Cool Check',sRcyText:='Unload From Wrong Slot (Board Quantity In Slot = 0).'),(sAlmText:='Board Capacity In Slot Is 0 While Unloading Buffer With Cool Check',sRcyText:='Unload From Wrong Slot (Board Capacity In Slot = 0).'),(sAlmText:='Unloading Slot Is Skipped While Unloading Buffer With Cool & Slot Check',sRcyText:='Unload From Wrong Slot (Skip Slot).'),(sAlmText:='Unloading Slot Is Not For Board While Unloading Buffer With Cool & Slot Check',sRcyText:='Unload From Wrong Slot (Not For Board).'),(sAlmText:='Unloading Slot Board Is Not available While Unloading Buffer With Cool & Slot Check',sRcyText:='Unload From Wrong Slot (Board Is Not Available).'),(sAlmText:='Unloading Last Sub Slot Is Not For Board While Unloading Buffer With Cool & Slot Check',sRcyText:='Unload From Wrong Slot (Last Sub Slot Is Not For Board).'),(sAlmText:='Unloading Last Sub Slot Has No Board While Unloading Buffer With Cool & Slot Check',sRcyText:='Unload From Wrong Slot (Last Sub Slot Has No Board).'),(sAlmText:='Board Quantity In Slot Is 0 While Unloading Buffer With Cool & Slot Check',sRcyText:='Unload From Wrong Slot (Board Quantity In Slot = 0).'),(sAlmText:='Board Capacity In Slot Is 0 While Unloading Buffer With Cool & Slot Check',sRcyText:='Unload From Wrong Slot (Board Capacity In Slot = 0).'),(sAlmText:='Loading Slot Is Not For Board',sRcyText:='Load To Wrong Slot (Not For Board).'),(sAlmText:='Loading Slot Is Full Of Board',sRcyText:='Load To Wrong Slot (Full With Board).'),(sAlmText:='Loading First Sub-Slot Is Not For Board',sRcyText:='Load To Wrong Slot (First Sub Slot Not For Board).'),(sAlmText:='Loading Last Sub-Slot Have Board, Which Mean Slot Is Full Of Board',sRcyText:='Load To Wrong Slot (Full With Board(Last Sub Slot Have Board)).'),(sAlmText:='Loading Last Sub-Slot Is Not For Board',sRcyText:='Load To Wrong Slot (Last Sub Slot Not For Board).'),(sAlmText:='Loading Slot Is Full Of Board',sRcyText:='Load To Wrong Slot (Full With Board).'),(sAlmText:='Loading Slot Is Skipped',sRcyText:='Load To Wrong Slot (Skip Slot).'),(sAlmText:='Existing Board Status Is Different With Loading Board Status',sRcyText:='Existing Board Status Is Different With Loading Buffer Status.'),(sAlmText:='Loading Slot Is Not For Board',sRcyText:='Load To Wrong Slot (Not For Board).'),(sAlmText:='Loading Slot Is Full Of Board',sRcyText:='Load To Wrong Slot (Full With Board).'),(sAlmText:='Loading First Sub-Slot Is Not For Board',sRcyText:='Load To Wrong Slot (First Sub Slot Not For Board).'),(sAlmText:='Loading Last Sub-Slot Have Board, Which Mean Slot Is Full Of Board',sRcyText:='Load To Wrong Slot (Full With Board(Last Sub Slot Have Board)).'),(sAlmText:='Loading Last Sub-Slot Is Not For Board',sRcyText:='Load To Wrong Slot (Last Sub Slot Not For Board).'),(sAlmText:='Loading Slot Is Full Of Board',sRcyText:='Load To Wrong Slot (Full With Board).'),(sAlmText:='Loading Slot Is Skipped',sRcyText:='Load To Wrong Slot (Skip Slot).'),(sAlmText:='Existing Board Status Is Different With Loading Board Status',sRcyText:='Existing Board Status Is Different With Loading Buffer Status.'),8((0))];
END_VAR
(**)
(*Local Output*)
VAR
	diNxtLoadSlt : DINT;
	diNxtUnloadSlt : DINT;
	diCoolBrdAny : DINT;
	diCoolBrdGd : DINT;
	diCoolBrdBad : DINT;
	bCoolNotRdy : BOOL;
	tyBuffer : tyBffr;
	tyDispBuffer : tyDispBffr;
	tyBufferStat : tyBffrStat;
	tyBoardUnloadStat : tyBrdUnloadStat;
	bFileNotFound : BOOL;
	bCoolFanCtrl : BOOL;
END_VAR
VAR RETAIN
	bMagPresent : BOOL;
END_VAR
VAR
	dtMagPresentTm : DATE_AND_TIME;
	bNewProduct : BOOL;
	bLastProductUnload : BOOL;
	bLastProductLeftInBffr : BOOL;
	bParamDiff : BOOL;
	bMagRemoved : BOOL;
	bFIFOOld : BOOL;
END_VAR
(**)
(*Local Input*)
VAR
	udiRstErr : UDINT := 0;
	sFileName : STRING[80] := 'Buffer.dat';
	bManual : BOOL := FALSE;
	dtCurrDT : DATE_AND_TIME;
	diMinSlt : DINT;
	diMaxSlt : DINT;
	diPitch : DINT;
	diSltCap : DINT := 1;
	diBffrTtlSlt : DINT;
	diCoolTm : DINT;
	diSltToSltInUM : DINT;
	diLifterBtmPosInUM : DINT;
	diLifterCurrPosInUM : DINT;
	bAscending : BOOL;
	bFIFO : BOOL;
	bGdBrdIn : BOOL;
	bGdBrdReq : BOOL;
	bNxtLoadSeq : BOOL;
	a_bSkip : ARRAY[1..c_diBffrSize] OF BOOL;
	diCoolFanOffDlyTm : DINT := 30000;
	bMagPresentSensor : BOOL;
	bPrepCoolFan : BOOL := TRUE;
	bCoolFanTm : BOOL := TRUE;
	sBffrNm : STRING[15];
	sProdNm : STRING[15];
	sBarcode1 : STRING[80];
	sBarcode2 : STRING[80];
	sCurrRcpNm : {REDUND_UNREPLICABLE} STRING[15];
	sProgNm : STRING[15] := 'Buffer';
	bNtSettingsLoadDone : BOOL := TRUE;
END_VAR
(**)
(*Local*)
VAR
	bRstErr : BOOL;
	udiRstErrOld : UDINT;
	bInitDone : BOOL;
	bInitialDone : BOOL;
	bUpdateSensor : BOOL;
	bBffrSetMty : BOOL;
	bBffrSetFull : BOOL;
	bUpdtDisplay : BOOL;
	usiStep : USINT;
	diCurrSlt : DINT;
	diExpectedSlt : DINT;
	bSetFull : BOOL;
	bSetMty : BOOL;
	bCoolFanRun : BOOL;
	tyBffrParameter : tyBffrParam;
	fbDirCreate1 : fbDirCreate;
	fbDirCreate2 : fbDirCreate;
	fbFileRead1 : fbFileFullRead;
	fbFileWrite1 : fbFileFullWrite;
	fbCoolFanOffDlyTm : TON;
	fbCoolFanOffChkTm : TON := (PT:=T#500ms);
	fbMagAbsentTm : TON := (PT:=T#5s);
	fbMagPresentTm : TON := (PT:=T#8s);
	eStatOld : eBufferAction := BufferActIdle;
	udiModuleNum : UDINT := 2001;
	diCurrSltHermes : DINT;
END_VAR
```

#### Act_Alarm.st
```iecst
(** 2019-03-25 **)
ACTION Act_Alarm:

	//Error
	IF EDGEPOS(eStatus = Error) THEN

		tyAlmData.sProgNm		:= p_sProgNm;
		tyAlmData.udiCode		:= udiStatus;
		tyAlmData.eSeverity		:= AlmSeverityError;
		tyAlmData.udiRunTime	:= tyAlmData.udiRunTime + 1;
		tyAlmData.bAlm			:= TRUE;
		tyAlmData.udiModuleNum  := udiModuleNum;
		g_sBufferProgNm		:= p_sProgNm;
		//Get Error Message
		IF tyAlmData.udiCode < 10000 OR tyAlmData.udiCode > 10099 THEN
			tyAlmData.sAlmMsg	:= 'Unknown';
			tyAlmData.sRcyMsg	:= 'Unknown';
		ELSE
			tyAlmData.sAlmMsg	:= a_tyAlmText[tyAlmData.udiCode].sAlmText;
			tyAlmData.sRcyMsg	:= a_tyAlmText[tyAlmData.udiCode].sRcyText;
		END_IF

		sStatTxt	:= tyAlmData.sAlmMsg;

	ELSIF bRstErr AND (tyAlmData.udiCode <> 0) THEN

		tyAlmData.udiCode	:= 0;
		tyAlmData.eSeverity	:= AlmSeverityNA;
		tyAlmData.sAlmMsg	:= '';
		tyAlmData.sRcyMsg	:= '';
		tyAlmData.bAlm			:= FALSE;
		sStatTxt	:= a_sStatText[eStat];

	END_IF

END_ACTION
```

#### Act_Background.st
```iecst
(** 2019-07-03 **)
ACTION Act_Background:

	fbMagPresentTm(IN := p_bMagPresentSensor);
	diCurrSltHermes	:= fLifterPosInUMToSltBtmMin(p_diLifterCurrPosInUM , p_diSltToSltInUM , p_diLifterBtmPosInUM);

	//Update Retain
	IF bUpdateSensor = TRUE THEN
		bMagPresent	:= fbMagPresentTm.Q;
	END_IF

	//Display Buffer
	IF bUpdtDisplay = TRUE THEN
		fDispBffrDescending(ADR(p_tyDispBuffer) , tyBffrParameter , p_tyBuffer , p_dtCurrDT , DINT_TO_TIME(p_diCoolTm) , 0 , 1 , 2);
	END_IF

	//Cooling Fan Control
	IF p_bManual = TRUE THEN
		;

	ELSIF bCoolFanRun = TRUE AND p_bPrepCoolFan = TRUE AND bCoolFanTm = TRUE THEN //Cooling Fan Control By Cooling Time

		fbCoolFanOffChkTm(IN := TRUE);

		IF fbCoolFanOffChkTm.Q = TRUE THEN
			IF fBffrChkCoolBrdAny(p_dtCurrDT, DINT_TO_TIME(p_diCoolTm), p_tyBuffer) = 0 THEN
				fbCoolFanOffDlyTm.IN	:= TRUE;
			ELSE
				fbCoolFanOffDlyTm.IN	:= FALSE;
				bCoolFanCtrl			:= TRUE;
			END_IF

			fbCoolFanOffChkTm(IN := FALSE);
		END_IF

		fbCoolFanOffDlyTm;

		IF fbCoolFanOffDlyTm.Q = TRUE THEN
			bCoolFanCtrl	:= FALSE;
		END_IF

	ELSIF bCoolFanRun = TRUE AND p_bPrepCoolFan = TRUE AND bCoolFanTm = FALSE THEN	//Cooling Fan Control By Buffer Empty
		fbCoolFanOffDlyTm(IN := p_tyBufferStat.bBffrMty);

		IF p_tyBufferStat.bBffrMty = FALSE THEN
			bCoolFanCtrl	:= TRUE;
		END_IF

		IF fbCoolFanOffDlyTm.Q = TRUE THEN
			bCoolFanCtrl	:= FALSE;
		END_IF

	ELSE

		bCoolFanCtrl	:= FALSE;

	END_IF

	//Set Buffer By Magazine Present
	IF bBffrSetFull = TRUE THEN
		IF p_bMagPresentSensor = TRUE AND fbMagAbsentTm.Q = TRUE THEN
			bSetFull		:= TRUE;
			dtMagPresentTm	:= p_dtCurrDT;
		END_IF

		IF bSetFull = TRUE THEN
			p_eAct	:= BufferActSetFull;

			IF eStatus = Done AND eStat = BufferActSetFull THEN
				p_eAct		:= BufferActIdle;
				bSetFull	:= FALSE;
			ELSIF eStatus = Error THEN
				bSetFull	:= FALSE;
			END_IF
		END_IF

		fbMagAbsentTm(IN := NOT p_bMagPresentSensor);

	ELSIF bBffrSetMty = TRUE THEN
		IF p_bMagPresentSensor = TRUE AND fbMagAbsentTm.Q = TRUE THEN
			bSetMty			:= TRUE;
			dtMagPresentTm	:= p_dtCurrDT;
		END_IF

		IF bSetMty = TRUE THEN
			p_eAct	:= BufferActSetMty;

			IF eStatus = Done AND eStat = BufferActSetMty THEN
				p_eAct	:= BufferActIdle;
				bSetMty	:= FALSE;
			ELSIF eStatus = Error THEN
				bSetMty	:= FALSE;
			END_IF
		END_IF

		fbMagAbsentTm(IN := NOT p_bMagPresentSensor);

	END_IF

	//Check Parameter Different
	bParamDiff	:= (tyBffrParameter.bAscending <> p_bAscending)
	OR (tyBffrParameter.diMinSlt <> p_diMinSlt)
	OR (tyBffrParameter.diMaxSlt <> p_diMaxSlt)
	OR (tyBffrParameter.diPitch <> p_diPitch)
	OR (tyBffrParameter.diSltCap <> p_diSltCap)
	OR (bFIFOOld <> p_bFIFO);

	//Update MagRemoved
	bMagRemoved	:= fbMagAbsentTm.Q;

END_ACTION
```

#### Act_InitGlobal.st
```iecst
(** 2019-04-26 **)
ACTION Act_InitGlobal:

	(* Always Change If Project Change *)

	//Pass Data To Link
	p_bLinkStartupRun ACCESS p_StartupRun;
	p_bLinkNtParamProjMagConvPrep ACCESS p_NtParamProjMag3ConvPrep;
//	p_eLinkOpsMagLDBufferAct ACCESS p_OpsMagLD3BufferAct;
	p_eLinkOpsMagConvLDBufferAct ACCESS p_OpsMagConvLD3BufferAct;

	p_bLinkMcParamProdSelTopToBtm ACCESS p_NtParamProjTopToBtmDefault;//p_ProdRcpCurrRcp1TopToBtm;
	p_bLinkPresentSen1 ACCESS p_DIMagPresentSen3;
	p_bLinkPresentSen2 ACCESS p_DIMagConvEntSen3;

	p_eLinkMag ACCESS p_NtParamProjMag;
	p_usiLinkMod ACCESS p_ProdRcpCurrRcp1McMod;

	p_diLinkSltToSltDist ACCESS p_MagRcpCurrRcpSltToSlt;
	p_diLinkMinSlt ACCESS p_ProdRcpCurrRcp1MinSltValue;
	p_diLinkMaxSlt ACCESS p_ProdRcpCurrRcp1MaxSltValue;
	p_diLinkPitch ACCESS p_ProdRcpCurrRcp1Pitch;
	p_diLinkBffrTtlSlt ACCESS p_MagRcpCurrRcpTtlSlt;
	p_diLinkLifterBtmPosInUM ACCESS p_MagRcpCurrRcpMag3Slt1Pos;

	p_diLinkSltToSltDist1 ACCESS p_MagRcpCurrRcpSltToSlt1;
	p_diLinkMinSlt1 ACCESS p_ProdRcpCurrRcp1MinSltRear;
	p_diLinkMaxSlt1 ACCESS p_ProdRcpCurrRcp1MaxSltRear;
	p_diLinkPitch1 ACCESS p_ProdRcpCurrRcp1PitchRear;
	p_diLinkBffrTtlSlt1 ACCESS p_MagRcpCurrRcpTtlSlt1;
	p_diLinkLifterBtmPosInUM1 ACCESS p_MagRcpCurrRcpMag3Slt1Pos1;

	p_bLinkNtParamProjRotCylPrep ACCESS p_NtParamProjPullerRotCylPrep;

	p_bLinkProjLifterMagPlatform ACCESS p_NtParamProjLifterMagPlatform;
	p_diNtParamProjMagMaxSlt ACCESS p_NtParamProjMagMaxSlt; //initial
	p_eLinkOpsLifMagLDBufferAct ACCESS p_OpsLifMagLDBufferAct3;
	p_bNtParamAutoRcpPrep ACCESS p_NtParamAutoRcpPrep;
	p_bHermesSvyPrep ACCESS p_NtParamHermesSvyPrep; //queryWO
	p_bMcParamHermesSvyEn ACCESS p_McParamHermesSvyEn;
	p_eNtParamCustomerReq ACCESS p_NtParamCustomerReq;
	p_bMcParamMesRFIDEn ACCESS p_McParamMesRFIDEn;

	//Pass Data To Internal Use
	p_udiRstErr ACCESS p_RstErrReset;
	p_sFileName ACCESS p_NtParamBffr3FileNm;
	p_bManual ACCESS p_UIMnlMod;
	p_dtCurrDT ACCESS p_TimeCurrDT;
//	p_diMinSlt ACCESS p_ProdRcpCurrRcp1MinSltValue;
//	p_diMaxSlt ACCESS p_ProdRcpCurrRcp1MaxSltValue;
//	p_diPitch ACCESS p_ProdRcpCurrRcp1Pitch;
//	p_diBffrTtlSlt ACCESS p_MagRcpCurrRcpTtlSlt;
//	p_diLifterBtmPosInUM ACCESS p_MagRcpCurrRcpMag3Slt1Pos;
	p_diLifterCurrPosInUM ACCESS p_LifterBtmActualPos;
	p_bFIFO ACCESS p_NtParamBffr3FIFO;
//	p_bMagPresentSensor ACCESS p_DIMagPresentSen3;
	p_sCurrRcpNm ACCESS p_ProdRcpCurrRcp1Nm;
	p_sProgNm ACCESS p_NtParamBffr3ProgNm;
	p_bNtSettingsLoadDone ACCESS p_StartupNtSettingsLoadDone;

	(* Always Change If Project Change *)

END_ACTION
```

#### Act_Initial.st
```iecst
(** 2019-04-26 **)
ACTION Act_Initial:

	//Initial
	sStatTxt	:= a_sStatText[eStat];

	fbDirCreate1.sDevice	:= 'F';
	fbDirCreate1.sDirName	:= 'User';
	fbDirCreate1(bEn := FALSE);

	fbDirCreate2.sDevice	:= 'User';
	fbDirCreate2.sDirName	:= 'Retain';
	fbDirCreate2(bEn := FALSE);

	fbFileRead1.sDevice			:= 'Retain';
	fbFileRead1.sFile			:= p_sFileName;
	fbFileRead1.udiOffset		:= 0;
	fbFileRead1.p_Dest			:= ADR(p_tyBuffer);
	fbFileRead1.udiLen			:= SIZEOF(p_tyBuffer);
	fbFileRead1(bEn := FALSE);

	fbFileWrite1.sDevice		:= 'Retain';
	fbFileWrite1.sFile			:= p_sFileName;
	fbFileWrite1.udiOffset		:= 0;
	fbFileWrite1.p_Src			:= ADR(p_tyBuffer);
	fbFileWrite1.udiLen			:= SIZEOF(p_tyBuffer);
	fbFileWrite1.udiOption		:= 0;
	fbFileWrite1(bEn := FALSE);

	fbCoolFanOffDlyTm.PT	:= DINT_TO_TIME(p_diCoolFanOffDlyTm);
	fbCoolFanOffDlyTm(IN := FALSE);

	fbCoolFanOffChkTm(IN := FALSE);
	fbMagAbsentTm(IN := FALSE);
	fbMagPresentTm(IN := FALSE);

	IF p_bLinkMcParamProdSelTopToBtm THEN
		diNxtUnloadSlt := 0;
	ELSE
		diNxtUnloadSlt := p_diNtParamProjMagMaxSlt;
	END_IF
END_ACTION
```

#### Act_Link.st
```iecst
(** 2019-03-29 **)
ACTION Act_Link:

	IF p_eLinkMag = LDMagQuadruple THEN
		CASE p_usiLinkMod OF
			0: //LDModLoadLnA:
				IF p_bAscending THEN
					p_diSltToSltInUM := p_diLinkSltToSltDist * -1;
				ELSE
					p_diSltToSltInUM := p_diLinkSltToSltDist;
				END_IF
				p_diMinSlt := p_diLinkMinSlt;
				p_diMaxSlt := p_diLinkMaxSlt;
				p_diPitch := p_diLinkPitch;
				p_diBffrTtlSlt := p_diLinkBffrTtlSlt;
				p_diLifterBtmPosInUM := p_diLinkLifterBtmPosInUM;

			1,2: //LDModLoadLnB, LDModLoadLnAB:
				IF p_bAscending THEN
					p_diSltToSltInUM := p_diLinkSltToSltDist1 * -1;
				ELSE
					p_diSltToSltInUM := p_diLinkSltToSltDist1;
				END_IF
				p_diMinSlt := p_diLinkMinSlt1;
				p_diMaxSlt := p_diLinkMaxSlt1;
				p_diPitch := p_diLinkPitch1;
				p_diBffrTtlSlt := p_diLinkBffrTtlSlt1;
				p_diLifterBtmPosInUM := p_diLinkLifterBtmPosInUM1;

		END_CASE
	ELSE
		IF p_bAscending THEN
			p_diSltToSltInUM := p_diLinkSltToSltDist * -1;
		ELSE
			p_diSltToSltInUM := p_diLinkSltToSltDist;
		END_IF
		IF p_bNtParamAutoRcpPrep AND ((p_bHermesSvyPrep AND p_bMcParamHermesSvyEn) OR (p_eNtParamCustomerReq = We_Fabricate AND p_bMcParamMesRFIDEn)) THEN
			p_diMinSlt ACCESS p_diAutoRcpMag3MinSlt;
			p_diMaxSlt ACCESS p_diAutoRcpMag3MaxSlt;
			p_diPitch ACCESS p_diAutoRcpMag3Pitch;
		ELSE
			p_diMinSlt ACCESS ADR(diMinSlt);
			p_diMaxSlt ACCESS ADR(diMaxSlt);
			p_diPitch ACCESS ADR(diPitch);
			p_diMinSlt := p_diLinkMinSlt;
			p_diMaxSlt := p_diLinkMaxSlt;
			p_diPitch := p_diLinkPitch;
		END_IF
		p_diBffrTtlSlt := p_diLinkBffrTtlSlt;
		p_diLifterBtmPosInUM := p_diLinkLifterBtmPosInUM;
	END_IF

	p_bAscending	:= NOT p_bLinkMcParamProdSelTopToBtm;
//	IF p_bLinkNtParamProjRotCylPrep THEN
//		p_bAscending := TRUE;
//	ELSE
//		p_bAscending := FALSE;
//	END_IF

	IF p_bLinkNtParamProjMagConvPrep THEN
		fbMagPresentTm.PT	:= T#2s;
	ELSE
		fbMagPresentTm.PT	:= T#8s;
	END_IF

	p_bMagPresentSensor := p_bLinkPresentSen1 OR p_bLinkPresentSen2;

END_ACTION
```

#### Act_LinkAction.st
```iecst
(** 2019-05-10 **)
ACTION Act_LinkAction:

	IF p_bLinkStartupRun = TRUE THEN
		p_eAct ACCESS p_StartupBuffer3Act;
	ELSE
		IF eStatus = Idle THEN
			IF p_bLinkProjLifterMagPlatform = FALSE THEN
				IF p_eLinkOpsMagConvLDBufferAct <> BufferActIdle THEN
					p_eAct ACCESS p_OpsMagConvLD3BufferAct;
				ELSE
					p_eAct ACCESS p_UIBuffer3Act;
				END_IF
			ELSE
				IF p_eLinkOpsLifMagLDBufferAct <> BufferActIdle THEN
					p_eAct ACCESS p_OpsLifMagLDBufferAct3;
				ELSE
					p_eAct ACCESS p_UIBuffer3Act;
				END_IF
			END_IF
		END_IF
	END_IF

END_ACTION
```

#### Act_Main.st
```iecst
(** 2019-07-03 **)
ACTION Act_Main:

	IF eStatOld <> eStat THEN
		fbDirCreate1(bEn := FALSE);
		fbDirCreate2(bEn := FALSE);
		fbFileRead1(bEn := FALSE);
		fbFileWrite1(bEn := FALSE);
		usiStep	:= 0;

		bFileNotFound			:= FALSE;
		bNewProduct				:= FALSE;
		bLastProductUnload		:= FALSE;
		bLastProductLeftInBffr	:= FALSE;

		sStatTxt	:= a_sStatText[eStat];

		eStatOld	:= eStat;

		eStatus		:= Busy;
	END_IF

	//Main
	CASE eStat OF

		BufferActIdle:
			eStatus	:= Idle;

		BufferActCreateDir:
			IF eStatus = Idle OR eStatus = Busy THEN

				eStatus	:= Busy;

				CASE usiStep OF
					0:
						fbDirCreate1(bEn := TRUE);
						IF fbDirCreate1.udiStatus = 0 THEN
							usiStep	:= 1;
						ELSIF fbDirCreate1.udiStatus < 65534 THEN
							eStatus		:= Error;

							IF fbDirCreate1.udiStatus = 1908 THEN
								udiStatus	:= 10000;	//Create User Directory Error
							ELSE
								udiStatus	:= fbDirCreate1.udiStatus;
							END_IF
						END_IF

					1:
						fbDirCreate2(bEn := TRUE);
						IF fbDirCreate2.udiStatus = 0 THEN
							eStatus	:= Done;
						ELSIF fbDirCreate2.udiStatus < 65534 THEN
							eStatus		:= Error;

							IF fbDirCreate2.udiStatus = 1908 THEN
								udiStatus	:= 10001;	//Create Retain Directory Error
							ELSE
								udiStatus	:= fbDirCreate2.udiStatus;
							END_IF
						END_IF

				END_CASE

			END_IF

		BufferActGetRetainBffr:
			IF eStatus = Idle OR eStatus = Busy THEN

				eStatus	:= Busy;

				fbFileRead1(bEn := TRUE);
				IF fbFileRead1.udiStatus = 0 THEN
					eStatus	:= Done;

					tyBffrParameter.diBffrTtlSlt	:= p_diBffrTtlSlt;
					tyBffrParameter.diSltCap		:= p_diSltCap;

					fBffrStat(ADR(p_tyBufferStat) , p_tyBuffer);
					fDispBffrDescending(ADR(p_tyDispBuffer) , tyBffrParameter , p_tyBuffer , p_dtCurrDT , DINT_TO_TIME(p_diCoolTm) , 0 , 1 , 2);

				ELSIF fbFileRead1.udiStatus < 65534 THEN
					eStatus	:= Error;

					IF fbFileRead1.udiStatus = 1900 THEN
						udiStatus	:= 10002;	//File Open Error While Reading Retain File
					ELSIF fbFileRead1.udiStatus = 1902 THEN
						udiStatus	:= 10003;	//File Read Error While Reading Retain File
					ELSIF fbFileRead1.udiStatus = 1904 THEN
						udiStatus	:= 10004;	//File Close Error While Reading Retain File
					ELSIF fbFileRead1.udiStatus = 1915 THEN
						eStatus			:= Done;
						bFileNotFound	:= TRUE;
					ELSE
						udiStatus	:= fbFileRead1.udiStatus;
					END_IF
				END_IF

			END_IF

		BufferActSetFull:
			IF eStatus = Idle OR eStatus = Busy THEN

				eStatus	:= Busy;

				CASE usiStep OF
					0:
						tyBffrParameter.bAscending		:= p_bAscending;
						tyBffrParameter.diBffrTtlSlt	:= p_diBffrTtlSlt;
						tyBffrParameter.diMaxSlt		:= p_diMaxSlt;
						tyBffrParameter.diMinSlt		:= p_diMinSlt;
						tyBffrParameter.diPitch			:= p_diPitch;
						tyBffrParameter.diSltCap		:= p_diSltCap;
						tyBffrParameter.a_bSkip			:= pa_bSkip;
						bFIFOOld						:= p_bFIFO;

						udiStatus	:= fBffrSetFull(ADR(p_tyBuffer) , tyBffrParameter , p_dtCurrDT , p_sBffrNm , p_sProdNm);

						IF udiStatus = 0 THEN
							usiStep	:= 1;

							fBffrStat(ADR(p_tyBufferStat) , p_tyBuffer);
							fDispBffrDescending(ADR(p_tyDispBuffer) , tyBffrParameter , p_tyBuffer , p_dtCurrDT , DINT_TO_TIME(p_diCoolTm) , 0 , 1 , 2);

						ELSE
							eStatus	:= Error;

						END_IF

					1:
						fbFileWrite1(bEn := TRUE);

						IF fbFileWrite1.udiStatus = 0 THEN
							eStatus	:= Done;
						ELSIF fbFileWrite1.udiStatus < 65534 THEN
							eStatus	:= Error;

							IF fbFileWrite1.udiStatus = 1900 THEN
								udiStatus	:= 10005;	//File Open Error While Setting Full Buffer
							ELSIF fbFileWrite1.udiStatus = 1901 THEN
								udiStatus	:= 10006;	//File Create Error While Setting Full Buffer
							ELSIF fbFileWrite1.udiStatus = 1903 THEN
								udiStatus	:= 10007;	//File Write Error While Setting Full Buffer
							ELSIF fbFileWrite1.udiStatus = 1904 THEN
								udiStatus	:= 10008;	//File Close Error While Setting Full Buffer
							ELSIF fbFileWrite1.udiStatus = 1914 THEN
								udiStatus	:= 10040;	//Directory Does Not Exist While Setting Full Buffer
							ELSE
								udiStatus	:= fbFileWrite1.udiStatus;
							END_IF
						END_IF

				END_CASE

			END_IF

		BufferActSetMty:
			IF eStatus = Idle OR eStatus = Busy THEN

				eStatus	:= Busy;

				CASE usiStep OF
					0:
						tyBffrParameter.bAscending		:= p_bAscending;
						tyBffrParameter.diBffrTtlSlt	:= p_diBffrTtlSlt;
						tyBffrParameter.diMaxSlt		:= p_diMaxSlt;
						tyBffrParameter.diMinSlt		:= p_diMinSlt;
						tyBffrParameter.diPitch			:= p_diPitch;
						tyBffrParameter.diSltCap		:= p_diSltCap;
						tyBffrParameter.a_bSkip			:= pa_bSkip;
						bFIFOOld						:= p_bFIFO;

						udiStatus	:= fBffrSetMty(ADR(p_tyBuffer) , tyBffrParameter , p_sBffrNm);

						IF udiStatus = 0 THEN
							usiStep	:= 1;

							fBffrStat(ADR(p_tyBufferStat) , p_tyBuffer);
							fDispBffrDescending(ADR(p_tyDispBuffer) , tyBffrParameter , p_tyBuffer , p_dtCurrDT , DINT_TO_TIME(p_diCoolTm) , 0 , 1 , 2);

						ELSE
							eStatus	:= Error;

						END_IF

					1:
						fbFileWrite1(bEn := TRUE);

						IF fbFileWrite1.udiStatus = 0 THEN
							eStatus	:= Done;
						ELSIF fbFileWrite1.udiStatus < 65534 THEN
							eStatus	:= Error;

							IF fbFileWrite1.udiStatus = 1900 THEN
								udiStatus	:= 10009;	//File Open Error While Setting Empty Buffer
							ELSIF fbFileWrite1.udiStatus = 1901 THEN
								udiStatus	:= 10010;	//File Create Error While Setting Empty Buffer
							ELSIF fbFileWrite1.udiStatus = 1903 THEN
								udiStatus	:= 10011;	//File Write Error While Setting Empty Buffer
							ELSIF fbFileWrite1.udiStatus = 1904 THEN
								udiStatus	:= 10012;	//File Close Error While Setting Empty Buffer
							ELSIF fbFileWrite1.udiStatus = 1914 THEN
								udiStatus	:= 10041;	//Directory Does Not Exist While Setting Empty Buffer
							ELSE
								udiStatus	:= fbFileWrite1.udiStatus;
							END_IF
						END_IF

				END_CASE

			END_IF

		BufferActLoad:
			IF eStatus = Idle OR eStatus = Busy THEN

				eStatus	:= Busy;

				CASE usiStep OF
					0:
						diCurrSlt	:= fLifterPosInUMToSltBtmMin(p_diLifterCurrPosInUM , p_diSltToSltInUM , p_diLifterBtmPosInUM);

						udiStatus	:= fBffrLoad(ADR(p_tyBuffer) , ADR(bNewProduct) , diCurrSlt , p_dtCurrDT , p_bGdBrdIn , p_sProdNm , p_sBarcode1 , p_sBarcode2);

						IF udiStatus = 0 THEN
							usiStep	:= 1;

							tyBffrParameter.diBffrTtlSlt	:= p_diBffrTtlSlt;
							tyBffrParameter.diSltCap		:= p_diSltCap;

							fBffrStat(ADR(p_tyBufferStat) , p_tyBuffer);
							fDispBffrDescending(ADR(p_tyDispBuffer) , tyBffrParameter , p_tyBuffer , p_dtCurrDT , DINT_TO_TIME(p_diCoolTm) , 0 , 1 , 2);

						ELSE
							eStatus	:= Error;

							IF udiStatus = 1010 THEN
								udiStatus	:= 10076;	//Loading Slot Is Not For Board
							ELSIF udiStatus = 1011 THEN
								udiStatus	:= 10077;	//Loading Slot Is Full Of Board
							ELSIF udiStatus = 1012 THEN
								udiStatus	:= 10078;	//Loading First Sub-Slot Is Not For Board
							ELSIF udiStatus	= 1013 THEN
								udiStatus	:= 10079;	//Loading Last Sub-Slot Have Board, Which Mean Slot Is Full Of Board
							ELSIF udiStatus = 1014 THEN
								udiStatus	:= 10080;	//Loading Last Sub-Slot Is Not For Board
							ELSIF udiStatus = 1015 THEN
								udiStatus	:= 10081;	//Loading Slot Is Full Of Board
							ELSIF udiStatus = 1001 THEN
								udiStatus	:= 10082;	//Loading Slot Is Skipped
							ELSIF udiStatus	= 1016 THEN
								udiStatus	:= 10083;	//Existing Board Status Is Different With Loading Board Status
							END_IF

						END_IF

					1:
						fbFileWrite1(bEn := TRUE);

						IF fbFileWrite1.udiStatus = 0 THEN
							eStatus	:= Done;
						ELSIF fbFileWrite1.udiStatus < 65534 THEN
							eStatus	:= Error;

							IF fbFileWrite1.udiStatus = 1900 THEN
								udiStatus	:= 10013;	//File Open Error While Loading Info To Buffer
							ELSIF fbFileWrite1.udiStatus = 1901 THEN
								udiStatus	:= 10014;	//File Create Error While Loading Info To Buffer
							ELSIF fbFileWrite1.udiStatus = 1903 THEN
								udiStatus	:= 10015;	//File Write Error While Loading Info To Buffer
							ELSIF fbFileWrite1.udiStatus = 1904 THEN
								udiStatus	:= 10016;	//File Close Error While Loading Info To Buffer
							ELSIF fbFileWrite1.udiStatus = 1914 THEN
								udiStatus	:= 10042;	//Directory Does Not Exist While Loading Info To Buffer
							ELSE
								udiStatus	:= fbFileWrite1.udiStatus;
							END_IF
						END_IF

				END_CASE

			END_IF

		BufferActLoadSltChk:
			IF eStatus = Idle OR eStatus = Busy THEN

				eStatus	:= Busy;

				CASE usiStep OF
					0:
						diCurrSlt	:= fLifterPosInUMToSltBtmMin(p_diLifterCurrPosInUM , p_diSltToSltInUM , p_diLifterBtmPosInUM);

						IF p_bNxtLoadSeq = TRUE AND p_bGdBrdIn = TRUE THEN
							diExpectedSlt	:= fBffrNxtLoadSeqGd(p_bAscending , p_tyBuffer);
						ELSIF p_bNxtLoadSeq = TRUE AND p_bGdBrdIn = FALSE THEN
							diExpectedSlt	:= fBffrNxtLoadSeqBad(p_bAscending , p_tyBuffer);
						ELSIF p_bNxtLoadSeq = FALSE AND p_bGdBrdIn = TRUE THEN
							diExpectedSlt	:= fBffrNxtLoadNearbyGd(diCurrSlt , p_tyBuffer);
						ELSE
							diExpectedSlt	:= fBffrNxtLoadNearbyBad(diCurrSlt , p_tyBuffer);
						END_IF

						IF diCurrSlt = diExpectedSlt THEN
							udiStatus	:= fBffrLoad(ADR(p_tyBuffer) , ADR(bNewProduct) , diCurrSlt , p_dtCurrDT , p_bGdBrdIn , p_sProdNm , p_sBarcode1 , p_sBarcode2);

							IF udiStatus = 0 THEN
								usiStep	:= 1;

								tyBffrParameter.diBffrTtlSlt	:= p_diBffrTtlSlt;
								tyBffrParameter.diSltCap		:= p_diSltCap;

								fBffrStat(ADR(p_tyBufferStat) , p_tyBuffer);
								fDispBffrDescending(ADR(p_tyDispBuffer) , tyBffrParameter , p_tyBuffer , p_dtCurrDT , DINT_TO_TIME(p_diCoolTm) , 0 , 1 , 2);

							ELSE
								eStatus	:= Error;

								IF udiStatus = 1010 THEN
									udiStatus	:= 10084;	//Loading Slot Is Not For Board
								ELSIF udiStatus = 1011 THEN
									udiStatus	:= 10085;	//Loading Slot Is Full Of Board
								ELSIF udiStatus = 1012 THEN
									udiStatus	:= 10086;	//Loading First Sub-Slot Is Not For Board
								ELSIF udiStatus	= 1013 THEN
									udiStatus	:= 10087;	//Loading Last Sub-Slot Have Board, Which Mean Slot Is Full Of Board
								ELSIF udiStatus = 1014 THEN
									udiStatus	:= 10088;	//Loading Last Sub-Slot Is Not For Board
								ELSIF udiStatus = 1015 THEN
									udiStatus	:= 10089;	//Loading Slot Is Full Of Board
								ELSIF udiStatus = 1001 THEN
									udiStatus	:= 10090;	//Loading Slot Is Skipped
								ELSIF udiStatus	= 1016 THEN
									udiStatus	:= 10091;	//Existing Board Status Is Different With Loading Board Status
								END_IF

							END_IF

						ELSE
							udiStatus	:= 10017;	//Wrong Slot Number To Load
							eStatus		:= Error;

						END_IF

					1:
						fbFileWrite1(bEn := TRUE);

						IF fbFileWrite1.udiStatus = 0 THEN
							eStatus	:= Done;
						ELSIF fbFileWrite1.udiStatus < 65534 THEN
							eStatus	:= Error;

							IF fbFileWrite1.udiStatus = 1900 THEN
								udiStatus	:= 10018;	//File Open Error While Loading Info To Buffer With Slot Check
							ELSIF fbFileWrite1.udiStatus = 1901 THEN
								udiStatus	:= 10019;	//File Create Error While Loading Info To Buffer With Slot Check
							ELSIF fbFileWrite1.udiStatus = 1903 THEN
								udiStatus	:= 10020;	//File Write Error While Loading Info To Buffer With Slot Check
							ELSIF fbFileWrite1.udiStatus = 1904 THEN
								udiStatus	:= 10021;	//File Close Error While Loading Info To Buffer With Slot Check
							ELSIF fbFileWrite1.udiStatus = 1914 THEN
								udiStatus	:= 10043;	//Directory Does Not Exist While Loading Info To Buffer With Slot Check
							ELSE
								udiStatus	:= fbFileWrite1.udiStatus;
							END_IF
						END_IF

				END_CASE

			END_IF

		BufferActUnload:
			IF eStatus = Idle OR eStatus = Busy THEN

				eStatus	:= Busy;

				CASE usiStep OF
					0:
						IF p_bLinkMcParamProdSelTopToBtm AND p_bLinkProjLifterMagPlatform = FALSE THEN //TravLif with Top to Btm
							diCurrSlt	:= fLifterPosInUMToSltTopMin(p_diLifterCurrPosInUM , p_diSltToSltInUM , p_diLifterBtmPosInUM);
						ELSE
							diCurrSlt	:= fLifterPosInUMToSltBtmMin(p_diLifterCurrPosInUM , p_diSltToSltInUM , p_diLifterBtmPosInUM);
						END_IF

						udiStatus	:= fBffrUnload(ADR(tyBoardUnloadStat) , ADR(p_tyBuffer) , ADR(bLastProductUnload) , ADR(bLastProductLeftInBffr) , diCurrSlt);

						IF p_sCurrRcpNm = tyBoardUnloadStat.sProdNm THEN
							bLastProductUnload	:= FALSE;
						END_IF

						IF udiStatus = 0 THEN
							usiStep	:= 1;

							tyBffrParameter.diBffrTtlSlt	:= p_diBffrTtlSlt;
							tyBffrParameter.diSltCap		:= p_diSltCap;

							fBffrStat(ADR(p_tyBufferStat) , p_tyBuffer);
							fDispBffrDescending(ADR(p_tyDispBuffer) , tyBffrParameter , p_tyBuffer , p_dtCurrDT , DINT_TO_TIME(p_diCoolTm) , 0 , 1 , 2);

						ELSE
							eStatus	:= Error;

							IF udiStatus = 1000 THEN
								udiStatus	:= 10048;	//Unloading Slot Is Skipped While Unloading Buffer
							ELSIF udiStatus = 1003 THEN
								udiStatus	:= 10049;	//Unloading Slot Is Not For Board While Unloading Buffer
							ELSIF udiStatus = 1004 THEN
								udiStatus	:= 10050;	//Unloading Slot Board Is Not available While Unloading Buffer
							ELSIF udiStatus = 1005 THEN
								udiStatus	:= 10051;	//Unloading Last Sub Slot Is Not For Board While Unloading Buffer
							ELSIF udiStatus = 1006 THEN
								udiStatus	:= 10052;	//Unloading Last Sub Slot Has No Board While Unloading Buffer
							ELSIF udiStatus = 1007 THEN
								udiStatus	:= 10053;	//Board Quantity In Slot Is 0 While Unloading Buffer
							ELSIF udiStatus = 1008 THEN
								udiStatus	:= 10054;	//Board Capacity In Slot Is 0 While Unloading Buffer
							END_IF

						END_IF

					1:
						fbFileWrite1(bEn := TRUE);

						IF fbFileWrite1.udiStatus = 0 THEN
							eStatus	:= Done;
						ELSIF fbFileWrite1.udiStatus < 65534 THEN
							eStatus	:= Error;

							IF fbFileWrite1.udiStatus = 1900 THEN
								udiStatus	:= 10022;	//File Open Error While Unloading Info From Buffer
							ELSIF fbFileWrite1.udiStatus = 1901 THEN
								udiStatus	:= 10023;	//File Create Error While Unloading Info From Buffer
							ELSIF fbFileWrite1.udiStatus = 1903 THEN
								udiStatus	:= 10024;	//File Write Error While Unloading Info From Buffer
							ELSIF fbFileWrite1.udiStatus = 1904 THEN
								udiStatus	:= 10025;	//File Close Error While Unloading Info From Buffer
							ELSIF fbFileWrite1.udiStatus = 1914 THEN
								udiStatus	:= 10044;	//Directory Does Not Exist While Unloading Info From Buffer
							ELSE
								udiStatus	:= fbFileWrite1.udiStatus;
							END_IF
						END_IF

				END_CASE

			END_IF

		BufferActUnloadSltChk:
			IF eStatus = Idle OR eStatus = Busy THEN

				eStatus	:= Busy;

				CASE usiStep OF
					0:
						diCurrSlt	:= fLifterPosInUMToSltBtmMin(p_diLifterCurrPosInUM , p_diSltToSltInUM , p_diLifterBtmPosInUM);

						IF p_bFIFO = TRUE AND p_bGdBrdReq = TRUE THEN
							diExpectedSlt	:= fBffrNxtUnloadFIFOGd(p_tyBuffer , '');
						ELSIF p_bFIFO = TRUE AND p_bGdBrdReq = FALSE THEN
							diExpectedSlt	:= fBffrNxtUnloadFIFOBad(p_tyBuffer , '');
						ELSIF p_bFIFO = FALSE AND p_bGdBrdReq = TRUE THEN
							diExpectedSlt	:= fBffrNxtUnloadLIFOGd(p_tyBuffer , '');
						ELSE
							diExpectedSlt	:= fBffrNxtUnloadLIFOBad(p_tyBuffer , '');
						END_IF

						IF diCurrSlt = diExpectedSlt THEN
							udiStatus	:= fBffrUnload(ADR(tyBoardUnloadStat) , ADR(p_tyBuffer) , ADR(bLastProductUnload) , ADR(bLastProductLeftInBffr) , diCurrSlt);

							IF p_sCurrRcpNm = tyBoardUnloadStat.sProdNm THEN
								bLastProductUnload	:= FALSE;
							END_IF

							IF udiStatus = 0 THEN
								usiStep	:= 1;

								tyBffrParameter.diBffrTtlSlt	:= p_diBffrTtlSlt;
								tyBffrParameter.diSltCap		:= p_diSltCap;

								fBffrStat(ADR(p_tyBufferStat) , p_tyBuffer);
								fDispBffrDescending(ADR(p_tyDispBuffer) , tyBffrParameter , p_tyBuffer , p_dtCurrDT , DINT_TO_TIME(p_diCoolTm) , 0 , 1 , 2);

							ELSE
								eStatus	:= Error;

								IF udiStatus = 1000 THEN
									udiStatus	:= 10055;	//Unloading Slot Is Skipped While Unloading Buffer With Slot Check
								ELSIF udiStatus = 1003 THEN
									udiStatus	:= 10056;	//Unloading Slot Is Not For Board While Unloading Buffer With Slot Check
								ELSIF udiStatus = 1004 THEN
									udiStatus	:= 10057;	//Unloading Slot Board Is Not available While Unloading Buffer With Slot Check
								ELSIF udiStatus = 1005 THEN
									udiStatus	:= 10058;	//Unloading Last Sub Slot Is Not For Board While Unloading Buffer With Slot Check
								ELSIF udiStatus = 1006 THEN
									udiStatus	:= 10059;	//Unloading Last Sub Slot Has No Board While Unloading Buffer With Slot Check
								ELSIF udiStatus = 1007 THEN
									udiStatus	:= 10060;	//Board Quantity In Slot Is 0 While Unloading Buffer With Slot Check
								ELSIF udiStatus = 1008 THEN
									udiStatus	:= 10061;	//Board Capacity In Slot Is 0 While Unloading Buffer With Slot Check
								END_IF

							END_IF

						ELSE
							udiStatus	:= 10026;	//Wrong Slot Number To Unload
							eStatus		:= Error;

						END_IF

					1:
						fbFileWrite1(bEn := TRUE);

						IF fbFileWrite1.udiStatus = 0 THEN
							eStatus	:= Done;
						ELSIF fbFileWrite1.udiStatus < 65534 THEN
							eStatus	:= Error;

							IF fbFileWrite1.udiStatus = 1900 THEN
								udiStatus	:= 10027;	//File Open Error While Unloading Info From Buffer With Slot Check
							ELSIF fbFileWrite1.udiStatus = 1901 THEN
								udiStatus	:= 10028;	//File Create Error While Unloading Info From Buffer With Slot Check
							ELSIF fbFileWrite1.udiStatus = 1903 THEN
								udiStatus	:= 10029;	//File Write Error While Unloading Info From Buffer With Slot Check
							ELSIF fbFileWrite1.udiStatus = 1904 THEN
								udiStatus	:= 10030;	//File Close Error While Unloading Info From Buffer With Slot Check
							ELSIF fbFileWrite1.udiStatus = 1914 THEN
								udiStatus	:= 10045;	//Directory Does Not Exist While Unloading Info From Buffer With Slot Check
							ELSE
								udiStatus	:= fbFileWrite1.udiStatus;
							END_IF
						END_IF

				END_CASE

			END_IF

		BufferActUnloadCoolChk:
			IF eStatus = Idle OR eStatus = Busy THEN

				eStatus	:= Busy;

				CASE usiStep OF
					0:
						diCurrSlt	:= fLifterPosInUMToSltBtmMin(p_diLifterCurrPosInUM , p_diSltToSltInUM , p_diLifterBtmPosInUM);

						bCoolNotRdy	:= NOT fBffrChkCoolTmRdy(diCurrSlt, p_dtCurrDT, DINT_TO_TIME(p_diCoolTm), p_tyBuffer);

						IF bCoolNotRdy = FALSE THEN
							udiStatus	:= fBffrUnload(ADR(tyBoardUnloadStat) , ADR(p_tyBuffer) , ADR(bLastProductUnload) , ADR(bLastProductLeftInBffr) , diCurrSlt);

							IF p_sCurrRcpNm = tyBoardUnloadStat.sProdNm THEN
								bLastProductUnload	:= FALSE;
							END_IF

							IF udiStatus = 0 THEN
								usiStep	:= 1;

								tyBffrParameter.diBffrTtlSlt	:= p_diBffrTtlSlt;
								tyBffrParameter.diSltCap		:= p_diSltCap;

								fBffrStat(ADR(p_tyBufferStat) , p_tyBuffer);
								fDispBffrDescending(ADR(p_tyDispBuffer) , tyBffrParameter , p_tyBuffer , p_dtCurrDT , DINT_TO_TIME(p_diCoolTm) , 0 , 1 , 2);

							ELSE
								eStatus	:= Error;

								IF udiStatus = 1000 THEN
									udiStatus	:= 10062;	//Unloading Slot Is Skipped While Unloading Buffer With Cool Check
								ELSIF udiStatus = 1003 THEN
									udiStatus	:= 10063;	//Unloading Slot Is Not For Board While Unloading Buffer With Cool Check
								ELSIF udiStatus = 1004 THEN
									udiStatus	:= 10064;	//Unloading Slot Board Is Not available While Unloading Buffer With Cool Check
								ELSIF udiStatus = 1005 THEN
									udiStatus	:= 10065;	//Unloading Last Sub Slot Is Not For Board While Unloading Buffer With Cool Check
								ELSIF udiStatus = 1006 THEN
									udiStatus	:= 10066;	//Unloading Last Sub Slot Has No Board While Unloading Buffer With Cool Check
								ELSIF udiStatus = 1007 THEN
									udiStatus	:= 10067;	//Board Quantity In Slot Is 0 While Unloading Buffer With Cool Check
								ELSIF udiStatus = 1008 THEN
									udiStatus	:= 10068;	//Board Capacity In Slot Is 0 While Unloading Buffer With Cool Check
								END_IF

							END_IF

						ELSE
							eStatus	:= Done;

						END_IF

					1:
						fbFileWrite1(bEn := TRUE);

						IF fbFileWrite1.udiStatus = 0 THEN
							eStatus	:= Done;
						ELSIF fbFileWrite1.udiStatus < 65534 THEN
							eStatus	:= Error;

							IF fbFileWrite1.udiStatus = 1900 THEN
								udiStatus	:= 10031;	//File Open Error While Unloading Info From Buffer With Cooling Time Check
							ELSIF fbFileWrite1.udiStatus = 1901 THEN
								udiStatus	:= 10032;	//File Create Error While Unloading Info From Buffer With Cooling Time Check
							ELSIF fbFileWrite1.udiStatus = 1903 THEN
								udiStatus	:= 10033;	//File Write Error While Unloading Info From Buffer With Cooling Time Check
							ELSIF fbFileWrite1.udiStatus = 1904 THEN
								udiStatus	:= 10034;	//File Close Error While Unloading Info From Buffer With Cooling Time Check
							ELSIF fbFileWrite1.udiStatus = 1914 THEN
								udiStatus	:= 10046;	//Directory Does Not Exist While Unloading Info From Buffer With Cooling Time Check
							ELSE
								udiStatus	:= fbFileWrite1.udiStatus;
							END_IF
						END_IF

				END_CASE

			END_IF

		BufferActUnloadSltChkCoolChk:
			IF eStatus = Idle OR eStatus = Busy THEN

				eStatus	:= Busy;

				CASE usiStep OF
					0:
						diCurrSlt	:= fLifterPosInUMToSltBtmMin(p_diLifterCurrPosInUM , p_diSltToSltInUM , p_diLifterBtmPosInUM);

						IF p_bFIFO = TRUE AND p_bGdBrdReq = TRUE THEN
							diExpectedSlt	:= fBffrNxtUnloadFIFOGd(p_tyBuffer , '');
						ELSIF p_bFIFO = TRUE AND p_bGdBrdReq = FALSE THEN
							diExpectedSlt	:= fBffrNxtUnloadFIFOBad(p_tyBuffer , '');
						ELSIF p_bFIFO = FALSE AND p_bGdBrdReq = TRUE THEN
							diExpectedSlt	:= fBffrNxtUnloadLIFOGd(p_tyBuffer , '');
						ELSE
							diExpectedSlt	:= fBffrNxtUnloadLIFOBad(p_tyBuffer , '');
						END_IF

						IF diCurrSlt = diExpectedSlt THEN
							bCoolNotRdy	:= NOT fBffrChkCoolTmRdy(diCurrSlt, p_dtCurrDT, DINT_TO_TIME(p_diCoolTm), p_tyBuffer);

							IF bCoolNotRdy = FALSE THEN
								udiStatus	:= fBffrUnload(ADR(tyBoardUnloadStat) , ADR(p_tyBuffer) , ADR(bLastProductUnload) , ADR(bLastProductLeftInBffr) , diCurrSlt);

								IF p_sCurrRcpNm = tyBoardUnloadStat.sProdNm THEN
									bLastProductUnload	:= FALSE;
								END_IF

								IF udiStatus = 0 THEN
									usiStep	:= 1;

									tyBffrParameter.diBffrTtlSlt	:= p_diBffrTtlSlt;
									tyBffrParameter.diSltCap		:= p_diSltCap;

									fBffrStat(ADR(p_tyBufferStat) , p_tyBuffer);
									fDispBffrDescending(ADR(p_tyDispBuffer) , tyBffrParameter , p_tyBuffer , p_dtCurrDT , DINT_TO_TIME(p_diCoolTm) , 0 , 1 , 2);

								ELSE
									eStatus	:= Error;

									IF udiStatus = 1000 THEN
										udiStatus	:= 10069;	//Unloading Slot Is Skipped While Unloading Buffer With Cool & Slot Check
									ELSIF udiStatus = 1003 THEN
										udiStatus	:= 10070;	//Unloading Slot Is Not For Board While Unloading Buffer With Cool & Slot Check
									ELSIF udiStatus = 1004 THEN
										udiStatus	:= 10071;	//Unloading Slot Board Is Not available While Unloading Buffer With Cool & Slot Check
									ELSIF udiStatus = 1005 THEN
										udiStatus	:= 10072;	//Unloading Last Sub Slot Is Not For Board While Unloading Buffer With Cool & Slot Check
									ELSIF udiStatus = 1006 THEN
										udiStatus	:= 10073;	//Unloading Last Sub Slot Has No Board While Unloading Buffer With Cool & Slot Check
									ELSIF udiStatus = 1007 THEN
										udiStatus	:= 10074;	//Board Quantity In Slot Is 0 While Unloading Buffer With Cool & Slot Check
									ELSIF udiStatus = 1008 THEN
										udiStatus	:= 10075;	//Board Capacity In Slot Is 0 While Unloading Buffer With Cool & Slot Check
									END_IF

								END_IF

							ELSE
								eStatus	:= Done;

							END_IF

						ELSE
							udiStatus	:= 10035;	//Wrong Slot Number To Unload With Cooling Time Check
							eStatus		:= Error;

						END_IF

					1:
						fbFileWrite1(bEn := TRUE);

						IF fbFileWrite1.udiStatus = 0 THEN
							eStatus	:= Done;
						ELSIF fbFileWrite1.udiStatus < 65534 THEN
							eStatus	:= Error;

							IF fbFileWrite1.udiStatus = 1900 THEN
								udiStatus	:= 10036;	//File Open Error While Unloading Info From Buffer With Slot Check And Cooling Time Check
							ELSIF fbFileWrite1.udiStatus = 1901 THEN
								udiStatus	:= 10037;	//File Create Error While Unloading Info From Buffer With Slot Check And Cooling Time Check
							ELSIF fbFileWrite1.udiStatus = 1903 THEN
								udiStatus	:= 10038;	//File Write Error While Unloading Info From Buffer With Slot Check And Cooling Time Check
							ELSIF fbFileWrite1.udiStatus = 1904 THEN
								udiStatus	:= 10039;	//File Close Error While Unloading Info From Buffer With Slot Check And Cooling Time Check
							ELSIF fbFileWrite1.udiStatus = 1914 THEN
								udiStatus	:= 10047;	//Directory Does Not Exist While Unloading Info From Buffer With Slot Check And Cooling Time Check
							ELSE
								udiStatus	:= fbFileWrite1.udiStatus;
							END_IF
						END_IF

				END_CASE

			END_IF

		BufferActNxtLoad:
			IF eStatus = Idle OR eStatus = Busy THEN

				diCurrSlt	:= fLifterPosInUMToSltBtmMin(p_diLifterCurrPosInUM , p_diSltToSltInUM , p_diLifterBtmPosInUM);

				IF p_bNxtLoadSeq = TRUE THEN
					diNxtLoadSlt	:= fBffrNxtLoadSeqAny(p_bAscending , p_tyBuffer);
				ELSE
					diNxtLoadSlt	:= fBffrNxtLoadNearbyAny(diCurrSlt , p_tyBuffer);
				END_IF

				eStatus	:= Done;

			END_IF

		BufferActNxtLoadGd:
			IF eStatus = Idle OR eStatus = Busy THEN

				diCurrSlt	:= fLifterPosInUMToSltBtmMin(p_diLifterCurrPosInUM , p_diSltToSltInUM , p_diLifterBtmPosInUM);

				IF p_bNxtLoadSeq = TRUE THEN
					diNxtLoadSlt	:= fBffrNxtLoadSeqGd(p_bAscending , p_tyBuffer);
				ELSE
					diNxtLoadSlt	:= fBffrNxtLoadNearbyGd(diCurrSlt , p_tyBuffer);
				END_IF

				eStatus	:= Done;

			END_IF

		BufferActNxtLoadBad:
			IF eStatus = Idle OR eStatus = Busy THEN

				diCurrSlt	:= fLifterPosInUMToSltBtmMin(p_diLifterCurrPosInUM , p_diSltToSltInUM , p_diLifterBtmPosInUM);

				IF p_bNxtLoadSeq = TRUE THEN
					diNxtLoadSlt	:= fBffrNxtLoadSeqBad(p_bAscending , p_tyBuffer);
				ELSE
					diNxtLoadSlt	:= fBffrNxtLoadNearbyBad(diCurrSlt , p_tyBuffer);
				END_IF

				eStatus	:= Done;

			END_IF

		BufferActNxtUnload:
			IF eStatus = Idle OR eStatus = Busy THEN

				IF p_bFIFO = TRUE THEN
					diNxtUnloadSlt	:= fBffrNxtUnloadFIFOAny(p_tyBuffer , '');
				ELSE
					diNxtUnloadSlt	:= fBffrNxtUnloadLIFOAny(p_tyBuffer , '');
				END_IF

				eStatus	:= Done;

			END_IF

		BufferActNxtUnloadGd:
			IF eStatus = Idle OR eStatus = Busy THEN

				IF p_bFIFO = TRUE THEN
					diNxtUnloadSlt	:= fBffrNxtUnloadFIFOGd(p_tyBuffer , '');
				ELSE
					diNxtUnloadSlt	:= fBffrNxtUnloadLIFOGd(p_tyBuffer , '');
				END_IF

				eStatus	:= Done;

			END_IF

		BufferActNxtUnloadBad:
			IF eStatus = Idle OR eStatus = Busy THEN

				IF p_bFIFO = TRUE THEN
					diNxtUnloadSlt	:= fBffrNxtUnloadFIFOBad(p_tyBuffer , '');
				ELSE
					diNxtUnloadSlt	:= fBffrNxtUnloadLIFOBad(p_tyBuffer , '');
				END_IF

				eStatus	:= Done;

			END_IF

		BufferActChkCoolTm:
			diCurrSlt	:= fLifterPosInUMToSltBtmMin(p_diLifterCurrPosInUM , p_diSltToSltInUM , p_diLifterBtmPosInUM);

			bCoolNotRdy	:= NOT fBffrChkCoolTmRdy(diCurrSlt, p_dtCurrDT, DINT_TO_TIME(p_diCoolTm), p_tyBuffer);

			eStatus	:= Done;

		BufferActChkCoolBrdAny:
			diCoolBrdAny	:= fBffrChkCoolBrdAny(p_dtCurrDT, DINT_TO_TIME(p_diCoolTm), p_tyBuffer);

			eStatus	:= Done;

		BufferActChkCoolBrdGd:
			diCoolBrdGd		:= fBffrChkCoolBrdGd(p_dtCurrDT, DINT_TO_TIME(p_diCoolTm), p_tyBuffer);

			eStatus	:= Done;

		BufferActChkCoolBrdBad:
			diCoolBrdBad	:= fBffrChkCoolBrdBad(p_dtCurrDT, DINT_TO_TIME(p_diCoolTm), p_tyBuffer);

			eStatus	:= Done;

		BufferActRstBffr:
			IF eStatus = Idle OR eStatus = Busy THEN

				tyBffrParameter.diBffrTtlSlt	:= p_diBffrTtlSlt;
				tyBffrParameter.diSltCap		:= p_diSltCap;

				memset(ADR(p_tyBuffer) , 0 , SIZEOF(p_tyBuffer));
				fBffrStat(ADR(p_tyBufferStat) , p_tyBuffer);
				fDispBffrDescending(ADR(p_tyDispBuffer) , tyBffrParameter , p_tyBuffer , p_dtCurrDT , DINT_TO_TIME(p_diCoolTm) , 0 , 1 , 2);

				eStatus	:= Done;

			END_IF

		BufferActSetCoolFan:
			IF eStatus = Idle OR eStatus = Busy THEN

				bCoolFanCtrl	:= TRUE;
				eStatus			:= Done;

			END_IF

		BufferActRstCoolFan:
			IF eStatus = Idle OR eStatus = Busy THEN

				bCoolFanCtrl	:= FALSE;
				eStatus			:= Done;

			END_IF

		BufferActBGStartBffrSetFull:
			IF eStatus = Idle OR eStatus = Busy THEN

				bBffrSetFull	:= TRUE;
				bBffrSetMty		:= FALSE;
				eStatus			:= Done;

			END_IF

		BufferActBGStartBffrSetMty:
			IF eStatus = Idle OR eStatus = Busy THEN

				bBffrSetFull	:= FALSE;
				bBffrSetMty		:= TRUE;
				eStatus			:= Done;

			END_IF

		BufferActBGStopBffrSet:
			IF eStatus = Idle OR eStatus = Busy THEN

				bBffrSetFull	:= FALSE;
				bBffrSetMty		:= FALSE;
				eStatus			:= Done;

			END_IF

		BufferActBGStartUpdtSen:
			IF eStatus = Idle OR eStatus = Busy THEN

				bUpdateSensor	:= TRUE;
				eStatus			:= Done;

			END_IF

		BufferActBGStopUpdtSen:
			IF eStatus = Idle OR eStatus = Busy THEN

				bUpdateSensor	:= FALSE;
				eStatus			:= Done;

			END_IF

		BufferActBGStartUpdtDisplay:
			IF eStatus = Idle OR eStatus = Busy THEN

				bUpdtDisplay	:= TRUE;
				eStatus			:= Done;

			END_IF

		BufferActBGStopUpdtDisplay:
			IF eStatus = Idle OR eStatus = Busy THEN

				bUpdtDisplay	:= FALSE;
				eStatus			:= Done;

			END_IF

		BufferActBGStartCoolFan:
			IF eStatus = Idle OR eStatus = Busy THEN

				bCoolFanRun	:= TRUE;
				eStatus		:= Done;

			END_IF

		BufferActBGStopCoolFan:
			IF eStatus = Idle OR eStatus = Busy THEN

				bCoolFanRun	:= FALSE;
				eStatus		:= Done;

			END_IF

	END_CASE

END_ACTION
```

#### Init.st
```iecst
(** 2019-06-07 **)
PROGRAM _INIT

	(* Always Change If Project Change *)

	//Pass Address To Global Address For External Use
	//Action, State & Status
	p_Buffer3Stat		:= ADR(eStat);
	p_Buffer3Status		:= ADR(eStatus);
	p_Buffer3StatTxt	:= ADR(sStatTxt);

	//Alarm
	p_Buffer3AlmData	:= ADR(tyAlmData);

	//Output
	p_Buffer3NxtLoadSlt				:= ADR(diNxtLoadSlt);
	p_Buffer3NxtUnloadSlt			:= ADR(diNxtUnloadSlt);
	p_Buffer3CoolBrdAny				:= ADR(diCoolBrdAny);
	p_Buffer3CoolBrdGd				:= ADR(diCoolBrdGd);
	p_Buffer3CoolBrdBad				:= ADR(diCoolBrdBad);
	p_Buffer3CoolNotRdy				:= ADR(bCoolNotRdy);
	p_Buffer3Bffr					:= ADR(tyBuffer);
	p_Buffer3DispBffr				:= ADR(tyDispBuffer);
	p_Buffer3BffrStat				:= ADR(tyBufferStat);
	p_Buffer3BrdUnloadStat			:= ADR(tyBoardUnloadStat);
	p_Buffer3FileNotFound			:= ADR(bFileNotFound);
	p_Buffer3CoolFanCtrl			:= ADR(bCoolFanCtrl);
	p_Buffer3MagPresent				:= ADR(bMagPresent);
	p_Buffer3MagPresentTm			:= ADR(dtMagPresentTm);
	p_Buffer3NewProduct				:= ADR(bNewProduct);
	p_Buffer3LastProductUnload		:= ADR(bLastProductUnload);
	p_Buffer3LastProductLeftInBffr	:= ADR(bLastProductLeftInBffr);
	p_Buffer3ParamDiff				:= ADR(bParamDiff);
	p_Buffer3MagRemoved				:= ADR(bMagRemoved);
	p_Buffer3FIFOOld				:= ADR(bFIFOOld);

	//Svy Hermes
	p_Buffer3SlotNo					:= ADR(diCurrSltHermes);

	(* Always Change If Project Change *)

END_PROGRAM
```

### Buffer4.var - Change By Project
```iecst
(*2019-03-25*)
(**)
(*Action & State & Status*)
VAR
	p_Buffer4Stat : UDINT;
	p_Buffer4Status : UDINT;
	p_Buffer4StatTxt : UDINT;
END_VAR
(**)
(*Alarm*)
VAR
	p_Buffer4AlmData : UDINT;
END_VAR
(**)
(*Output*)
VAR
	p_Buffer4NxtLoadSlt : UDINT;
	p_Buffer4NxtUnloadSlt : UDINT;
	p_Buffer4CoolBrdAny : UDINT;
	p_Buffer4CoolBrdGd : UDINT;
	p_Buffer4CoolBrdBad : UDINT;
	p_Buffer4CoolNotRdy : UDINT;
	p_Buffer4Bffr : UDINT;
	p_Buffer4DispBffr : UDINT;
	p_Buffer4BffrStat : UDINT;
	p_Buffer4BrdUnloadStat : UDINT;
	p_Buffer4FileNotFound : UDINT;
	p_Buffer4CoolFanCtrl : UDINT;
	p_Buffer4MagPresent : UDINT;
	p_Buffer4MagPresentTm : UDINT;
	p_Buffer4NewProduct : UDINT;
	p_Buffer4LastProductUnload : UDINT;
	p_Buffer4LastProductLeftInBffr : UDINT;
	p_Buffer4ParamDiff : UDINT;
	p_Buffer4MagRemoved : UDINT;
	p_Buffer4FIFOOld : UDINT;
END_VAR
```

### Program Logical/Buffer/Buffer4 (IEC) - 1.00.0 - NtBuffer v5.00.0 , NtFileIO v5.00.0

#### InputRef_Link.var
```iecst
(*2019-04-09*)
(**)
(*External*)
VAR
	p_bLinkStartupRun : REFERENCE TO BOOL;
	p_bLinkNtParamProjMagConvPrep : REFERENCE TO BOOL;
	p_eLinkOpsMagLDBufferAct : REFERENCE TO eBufferAction;
	p_eLinkOpsMagConvLDBufferAct : REFERENCE TO eBufferAction;
END_VAR
(**)
VAR
	p_diLinkSltToSltDist : REFERENCE TO DINT;
	p_bLinkMcParamProdSelTopToBtm : REFERENCE TO BOOL;
	p_bLinkPresentSen1 : REFERENCE TO BOOL;
	p_bLinkPresentSen2 : REFERENCE TO BOOL;
END_VAR
(**)
VAR
	p_eLinkMag : REFERENCE TO eLDMag;
	p_usiLinkMod : REFERENCE TO USINT;
END_VAR
(**)
VAR
	p_diLinkMinSlt : REFERENCE TO DINT;
	p_diLinkMaxSlt : REFERENCE TO DINT;
	p_diLinkPitch : REFERENCE TO DINT;
	p_diLinkBffrTtlSlt : REFERENCE TO DINT;
	p_diLinkLifterBtmPosInUM : REFERENCE TO DINT;
END_VAR
(**)
VAR
	p_diLinkSltToSltDist1 : REFERENCE TO DINT;
	p_diLinkMinSlt1 : REFERENCE TO DINT;
	p_diLinkMaxSlt1 : REFERENCE TO DINT;
	p_diLinkPitch1 : REFERENCE TO DINT;
	p_diLinkBffrTtlSlt1 : REFERENCE TO DINT;
	p_diLinkLifterBtmPosInUM1 : REFERENCE TO DINT;
	p_bLinkNtParamProjRotCylPrep : REFERENCE TO BOOL;
END_VAR
(**)
VAR
	p_bLinkProjLifterMagPlatform : REFERENCE TO BOOL;
	p_eLinkOpsLifMagULBufferAct : REFERENCE TO eBufferAction;
	p_diNtParamProjMagMaxSlt : REFERENCE TO DINT;
END_VAR
```
